    |   movel([0.186644, -1.304676, -2.622886, -0.784827, 1.570796, 1.757440],accel_mss,speed_ms,0,blend_radius_m)
    |   movel([0.187241, -1.304577, -2.622946, -0.784867, 1.570796, 1.758037],accel_mss,speed_ms,0,blend_radius_m)
    |   movel([0.187800, -1.304513, -2.622984, -0.784892, 1.570796, 1.758596],accel_mss,speed_ms,0,blend_radius_m)
    |   movel([0.187953, -1.304694, -2.622875, -0.784820, 1.570796, 1.758749],accel_mss,speed_ms,0,blend_radius_m)
    |   movel([0.187710, -1.304999, -2.622692, -0.784698, 1.570796, 1.758506],accel_mss,speed_ms,0,blend_radius_m)
    |   movel([0.187182, -1.305200, -2.622571, -0.784618, 1.570796, 1.757979],accel_mss,speed_ms,0,blend_radius_m)
    |   movel([0.186600, -1.305390, -2.622457, -0.784543, 1.570796, 1.757397],accel_mss,speed_ms,0,blend_radius_m)
    |   movel([0.185739, -1.305642, -2.622305, -0.784442, 1.570796, 1.756535],accel_mss,speed_ms,0,blend_radius_m)
    |   movel([0.184876, -1.305876, -2.622164, -0.784349, 1.570796, 1.755672],accel_mss,speed_ms,0,blend_radius_m)
    |   movel([0.180549, -1.306967, -2.621506, -0.783916, 1.570796, 1.751345],accel_mss,speed_ms,0,blend_radius_m)
    |   movel([0.180549, -1.272923, -2.604715, -0.834751, 1.570796, 1.751345],accel_mss,speed_ms,0,blend_radius_m)
    |   speed_ms = 1.000
    |   movel([0.180846, -1.271403, -2.605588, -0.835398, 1.570796, 1.751642],accel_mss,speed_ms,0,blend_radius_m)
    |   speed_ms = 0.008
    |   movel([0.180846, -1.299028, -2.619389, -0.793972, 1.570796, 1.751642],accel_mss,speed_ms,0,blend_radius_m)
    |   speed_ms = 0.003
    |   movel([0.180846, -1.302530, -2.621035, -0.788824, 1.570796, 1.751642],accel_mss,speed_ms,0,blend_radius_m)
    |   speed_ms = 0.008
    |   movel([0.176518, -1.303606, -2.620389, -0.788394, 1.570796, 1.747315],accel_mss,speed_ms,0,blend_radius_m)
    |   movel([0.175664, -1.303803, -2.620271, -0.788315, 1.570796, 1.746460],accel_mss,speed_ms,0,blend_radius_m)
    |   movel([0.174818, -1.303978, -2.620165, -0.788245, 1.570796, 1.745615],accel_mss,speed_ms,0,blend_radius_m)
    |   movel([0.174256, -1.304075, -2.620107, -0.788207, 1.570796, 1.745053],accel_mss,speed_ms,0,blend_radius_m)
    |   movel([0.173758, -1.304132, -2.620073, -0.788184, 1.570796, 1.744555],accel_mss,speed_ms,0,blend_radius_m)
    |   movel([0.173618, -1.303922, -2.620199, -0.788268, 1.570796, 1.744415],accel_mss,speed_ms,0,blend_radius_m)
    |   movel([0.173863, -1.303642, -2.620367, -0.788379, 1.570796, 1.744659],accel_mss,speed_ms,0,blend_radius_m)
    |   movel([0.174452, -1.303418, -2.620502, -0.788469, 1.570796, 1.745248],accel_mss,speed_ms,0,blend_radius_m)
    |   movel([0.175069, -1.303213, -2.620625, -0.788551, 1.570796, 1.745865],accel_mss,speed_ms,0,blend_radius_m)
    |   movel([0.175893, -1.302967, -2.620773, -0.788649, 1.570796, 1.746689],accel_mss,speed_ms,0,blend_radius_m)
    |   movel([0.176718, -1.302738, -2.620910, -0.788741, 1.570796, 1.747515],accel_mss,speed_ms,0,blend_radius_m)
    |   movel([0.181025, -1.301632, -2.621573, -0.789184, 1.570796, 1.751821],accel_mss,speed_ms,0,blend_radius_m)
    |   movel([0.185323, -1.300575, -2.622205, -0.789610, 1.570796, 1.756120],accel_mss,speed_ms,0,blend_radius_m)
    |   movel([0.186140, -1.300389, -2.622315, -0.789685, 1.570796, 1.756936],accel_mss,speed_ms,0,blend_radius_m)
    |   movel([0.186952, -1.300226, -2.622412, -0.789750, 1.570796, 1.757748],accel_mss,speed_ms,0,blend_radius_m)
    |   movel([0.187550, -1.300126, -2.622472, -0.789791, 1.570796, 1.758346],accel_mss,speed_ms,0,blend_radius_m)
    |   movel([0.188109, -1.300062, -2.622510, -0.789816, 1.570796, 1.758906],accel_mss,speed_ms,0,blend_radius_m)
    |   movel([0.188263, -1.300243, -2.622402, -0.789743, 1.570796, 1.759059],accel_mss,speed_ms,0,blend_radius_m)
    |   movel([0.188019, -1.300551, -2.622219, -0.789619, 1.570796, 1.758815],accel_mss,speed_ms,0,blend_radius_m)
    |   movel([0.187491, -1.300752, -2.622099, -0.789538, 1.570796, 1.758287],accel_mss,speed_ms,0,blend_radius_m)
    |   movel([0.186908, -1.300943, -2.621985, -0.789461, 1.570796, 1.757704],accel_mss,speed_ms,0,blend_radius_m)
    |   movel([0.186045, -1.301196, -2.621833, -0.789359, 1.570796, 1.756841],accel_mss,speed_ms,0,blend_radius_m)
    |   movel([0.185180, -1.301432, -2.621692, -0.789265, 1.570796, 1.755976],accel_mss,speed_ms,0,blend_radius_m)
    |   movel([0.180846, -1.302530, -2.621035, -0.788824, 1.570796, 1.751642],accel_mss,speed_ms,0,blend_radius_m)
    |   movel([0.180846, -1.305477, -2.622404, -0.784508, 1.570796, 1.751642],accel_mss,speed_ms,0,blend_radius_m)
    |   movel([0.176518, -1.306551, -2.621757, -0.784081, 1.570796, 1.747315],accel_mss,speed_ms,0,blend_radius_m)
    |   movel([0.175664, -1.306747, -2.621638, -0.784003, 1.570796, 1.746460],accel_mss,speed_ms,0,blend_radius_m)
    |   movel([0.174818, -1.306923, -2.621532, -0.783934, 1.570796, 1.745615],accel_mss,speed_ms,0,blend_radius_m)
    |   movel([0.174256, -1.307019, -2.621474, -0.783896, 1.570796, 1.745053],accel_mss,speed_ms,0,blend_radius_m)
    |   movel([0.173758, -1.307076, -2.621440, -0.783873, 1.570796, 1.744555],accel_mss,speed_ms,0,blend_radius_m)
    |   movel([0.173618, -1.306867, -2.621566, -0.783956, 1.570796, 1.744415],accel_mss,speed_ms,0,blend_radius_m)
    |   movel([0.173863, -1.306587, -2.621735, -0.784067, 1.570796, 1.744659],accel_mss,speed_ms,0,blend_radius_m)
    |   movel([0.174452, -1.306364, -2.621870, -0.784155, 1.570796, 1.745248],accel_mss,speed_ms,0,blend_radius_m)
    |   movel([0.175069, -1.306159, -2.621993, -0.784237, 1.570796, 1.745865],accel_mss,speed_ms,0,blend_radius_m)
    |   movel([0.175893, -1.305913, -2.622141, -0.784334, 1.570796, 1.746689],accel_mss,speed_ms,0,blend_radius_m)
    |   movel([0.176718, -1.305685, -2.622279, -0.784425, 1.570796, 1.747515],accel_mss,speed_ms,0,blend_radius_m)
    |   movel([0.181025, -1.304581, -2.622943, -0.784865, 1.570796, 1.751821],accel_mss,speed_ms,0,blend_radius_m)
    |   movel([0.185323, -1.303526, -2.623577, -0.785287, 1.570796, 1.756120],accel_mss,speed_ms,0,blend_radius_m)
    |   movel([0.186140, -1.303340, -2.623688, -0.785361, 1.570796, 1.756936],accel_mss,speed_ms,0,blend_radius_m)
    |   movel([0.186952, -1.303178, -2.623785, -0.785426, 1.570796, 1.757748],accel_mss,speed_ms,0,blend_radius_m)
    |   movel([0.187550, -1.303078, -2.623845, -0.785466, 1.570796, 1.758346],accel_mss,speed_ms,0,blend_radius_m)
    |   movel([0.188109, -1.303014, -2.623883, -0.785492, 1.570796, 1.758906],accel_mss,speed_ms,0,blend_radius_m)
    |   movel([0.188263, -1.303195, -2.623775, -0.785419, 1.570796, 1.759059],accel_mss,speed_ms,0,blend_radius_m)
    |   movel([0.188019, -1.303501, -2.623591, -0.785297, 1.570796, 1.758815],accel_mss,speed_ms,0,blend_radius_m)
    |   movel([0.187491, -1.303702, -2.623471, -0.785216, 1.570796, 1.758287],accel_mss,speed_ms,0,blend_radius_m)
    |   movel([0.186908, -1.303893, -2.623356, -0.785140, 1.570796, 1.757704],accel_mss,speed_ms,0,blend_radius_m)
    |   movel([0.186045, -1.304146, -2.623204, -0.785039, 1.570796, 1.756841],accel_mss,speed_ms,0,blend_radius_m)
    |   movel([0.185180, -1.304381, -2.623063, -0.784945, 1.570796, 1.755976],accel_mss,speed_ms,0,blend_radius_m)
    |   movel([0.180846, -1.305477, -2.622404, -0.784508, 1.570796, 1.751642],accel_mss,speed_ms,0,blend_radius_m)
    |   movel([0.180846, -1.271403, -2.605588, -0.835398, 1.570796, 1.751642],accel_mss,speed_ms,0,blend_radius_m)
    |   speed_ms = 1.000
    |   movel([0.180878, -1.269658, -2.606587, -0.836144, 1.570796, 1.751674],accel_mss,speed_ms,0,blend_radius_m)
    |   speed_ms = 0.008
    |   movel([0.180878, -1.297310, -2.620412, -0.794668, 1.570796, 1.751674],accel_mss,speed_ms,0,blend_radius_m)
    |   speed_ms = 0.003
    |   movel([0.180878, -1.300815, -2.622061, -0.789513, 1.570796, 1.751674],accel_mss,speed_ms,0,blend_radius_m)
    |   speed_ms = 0.008
    |   movel([0.173221, -1.302766, -2.620894, -0.788730, 1.570796, 1.744017],accel_mss,speed_ms,0,blend_radius_m)
    |   movel([0.174123, -1.298088, -2.623685, -0.790616, 1.570796, 1.744920],accel_mss,speed_ms,0,blend_radius_m)
    |   movel([0.174373, -1.296883, -2.624400, -0.791107, 1.570796, 1.745169],accel_mss,speed_ms,0,blend_radius_m)
    |   movel([0.174623, -1.295770, -2.625057, -0.791561, 1.570796, 1.745419],accel_mss,speed_ms,0,blend_radius_m)
    |   movel([0.174967, -1.294373, -2.625881, -0.792134, 1.570796, 1.745763],accel_mss,speed_ms,0,blend_radius_m)
    |   movel([0.175412, -1.293345, -2.626486, -0.792558, 1.570796, 1.746208],accel_mss,speed_ms,0,blend_radius_m)
    |   movel([0.190492, -1.289495, -2.628739, -0.794155, 1.570796, 1.761288],accel_mss,speed_ms,0,blend_radius_m)
    |   movel([0.188541, -1.298906, -2.623199, -0.790284, 1.570796, 1.759338],accel_mss,speed_ms,0,blend_radius_m)
    |   movel([0.180878, -1.300815, -2.622061, -0.789513, 1.570796, 1.751674],accel_mss,speed_ms,0,blend_radius_m)
    |   movel([0.180878, -1.303765, -2.623433, -0.785191, 1.570796, 1.751674],accel_mss,speed_ms,0,blend_radius_m)
    |   movel([0.173221, -1.305712, -2.622262, -0.784414, 1.570796, 1.744017],accel_mss,speed_ms,0,blend_radius_m)
    |   movel([0.174123, -1.301044, -2.625060, -0.786285, 1.570796, 1.744920],accel_mss,speed_ms,0,blend_radius_m)
    |   movel([0.174373, -1.299841, -2.625777, -0.786772, 1.570796, 1.745169],accel_mss,speed_ms,0,blend_radius_m)
    |   movel([0.174623, -1.298730, -2.626436, -0.787222, 1.570796, 1.745419],accel_mss,speed_ms,0,blend_radius_m)
    |   movel([0.174967, -1.297336, -2.627262, -0.787791, 1.570796, 1.745763],accel_mss,speed_ms,0,blend_radius_m)
    |   movel([0.175412, -1.296309, -2.627869, -0.788211, 1.570796, 1.746208],accel_mss,speed_ms,0,blend_radius_m)
    |   movel([0.190492, -1.292466, -2.630127, -0.789796, 1.570796, 1.761288],accel_mss,speed_ms,0,blend_radius_m)
    |   movel([0.188541, -1.301860, -2.624573, -0.785956, 1.570796, 1.759338],accel_mss,speed_ms,0,blend_radius_m)
    |   movel([0.180878, -1.303765, -2.623433, -0.785191, 1.570796, 1.751674],accel_mss,speed_ms,0,blend_radius_m)
    |   movel([0.180878, -1.269658, -2.606587, -0.836144, 1.570796, 1.751674],accel_mss,speed_ms,0,blend_radius_m)
    |   speed_ms = 1.000
    |   movel([0.182720, -1.258496, -2.612890, -0.841002, 1.570796, 1.753516],accel_mss,speed_ms,0,blend_radius_m)
    |   speed_ms = 0.008
    |   movel([0.182720, -1.286315, -2.626867, -0.799207, 1.570796, 1.753516],accel_mss,speed_ms,0,blend_radius_m)
    |   speed_ms = 0.003
    |   movel([0.182720, -1.289844, -2.628536, -0.794009, 1.570796, 1.753516],accel_mss,speed_ms,0,blend_radius_m)
    |   speed_ms = 0.008
    |   movel([0.182439, -1.290140, -2.628363, -0.793886, 1.570796, 1.753235],accel_mss,speed_ms,0,blend_radius_m)
    |   movel([0.182079, -1.290336, -2.628249, -0.793804, 1.570796, 1.752875],accel_mss,speed_ms,0,blend_radius_m)
    |   movel([0.181259, -1.290643, -2.628069, -0.793676, 1.570796, 1.752055],accel_mss,speed_ms,0,blend_radius_m)
    |   movel([0.180843, -1.290767, -2.627997, -0.793625, 1.570796, 1.751639],accel_mss,speed_ms,0,blend_radius_m)
    |   movel([0.179595, -1.291104, -2.627800, -0.793485, 1.570796, 1.750391],accel_mss,speed_ms,0,blend_radius_m)
    |   movel([0.175569, -1.292152, -2.627186, -0.793050, 1.570796, 1.746365],accel_mss,speed_ms,0,blend_radius_m)
    |   movel([0.177282, -1.283292, -2.632329, -0.796768, 1.570796, 1.748078],accel_mss,speed_ms,0,blend_radius_m)
    |   movel([0.181054, -1.282298, -2.632900, -0.797191, 1.570796, 1.751850],accel_mss,speed_ms,0,blend_radius_m)
    |   movel([0.182542, -1.281936, -2.633107, -0.797346, 1.570796, 1.753338],accel_mss,speed_ms,0,blend_radius_m)
    |   movel([0.184186, -1.281601, -2.633299, -0.797489, 1.570796, 1.754982],accel_mss,speed_ms,0,blend_radius_m)
    |   movel([0.184431, -1.281745, -2.633217, -0.797427, 1.570796, 1.755227],accel_mss,speed_ms,0,blend_radius_m)
    |   movel([0.184458, -1.282004, -2.633069, -0.797317, 1.570796, 1.755254],accel_mss,speed_ms,0,blend_radius_m)
    |   movel([0.183920, -1.284771, -2.631478, -0.796141, 1.570796, 1.754716],accel_mss,speed_ms,0,blend_radius_m)
    |   movel([0.183450, -1.287114, -2.630123, -0.795152, 1.570796, 1.754246],accel_mss,speed_ms,0,blend_radius_m)
    |   movel([0.183040, -1.289069, -2.628987, -0.794333, 1.570796, 1.753836],accel_mss,speed_ms,0,blend_radius_m)
    |   movel([0.182907, -1.289456, -2.628762, -0.794171, 1.570796, 1.753704],accel_mss,speed_ms,0,blend_radius_m)
    |   movel([0.182720, -1.289844, -2.628536, -0.794009, 1.570796, 1.753516],accel_mss,speed_ms,0,blend_radius_m)
    |   movel([0.182720, -1.292815, -2.629923, -0.789651, 1.570796, 1.753516],accel_mss,speed_ms,0,blend_radius_m)
    |   movel([0.182439, -1.293111, -2.629750, -0.789529, 1.570796, 1.753235],accel_mss,speed_ms,0,blend_radius_m)
    |   movel([0.182079, -1.293306, -2.629635, -0.789448, 1.570796, 1.752875],accel_mss,speed_ms,0,blend_radius_m)
    |   movel([0.181259, -1.293613, -2.629455, -0.789321, 1.570796, 1.752055],accel_mss,speed_ms,0,blend_radius_m)
    |   movel([0.180843, -1.293736, -2.629383, -0.789270, 1.570796, 1.751639],accel_mss,speed_ms,0,blend_radius_m)
    |   movel([0.179595, -1.294072, -2.629186, -0.789131, 1.570796, 1.750391],accel_mss,speed_ms,0,blend_radius_m)
    |   movel([0.175569, -1.295119, -2.628570, -0.788700, 1.570796, 1.746365],accel_mss,speed_ms,0,blend_radius_m)
    |   movel([0.177282, -1.286275, -2.633726, -0.792388, 1.570796, 1.748078],accel_mss,speed_ms,0,blend_radius_m)
    |   movel([0.181054, -1.285283, -2.634298, -0.792808, 1.570796, 1.751850],accel_mss,speed_ms,0,blend_radius_m)
    |   movel([0.182542, -1.284921, -2.634506, -0.792961, 1.570796, 1.753338],accel_mss,speed_ms,0,blend_radius_m)
    |   movel([0.184186, -1.284587, -2.634699, -0.793104, 1.570796, 1.754982],accel_mss,speed_ms,0,blend_radius_m)
    |   movel([0.184431, -1.284730, -2.634616, -0.793043, 1.570796, 1.755227],accel_mss,speed_ms,0,blend_radius_m)
    |   movel([0.184458, -1.284989, -2.634467, -0.792933, 1.570796, 1.755254],accel_mss,speed_ms,0,blend_radius_m)
    |   movel([0.183920, -1.287751, -2.632873, -0.791766, 1.570796, 1.754716],accel_mss,speed_ms,0,blend_radius_m)
    |   movel([0.183450, -1.290090, -2.631514, -0.790785, 1.570796, 1.754246],accel_mss,speed_ms,0,blend_radius_m)
    |   movel([0.183040, -1.292042, -2.630376, -0.789972, 1.570796, 1.753836],accel_mss,speed_ms,0,blend_radius_m)
    |   movel([0.182907, -1.292427, -2.630150, -0.789812, 1.570796, 1.753704],accel_mss,speed_ms,0,blend_radius_m)
    |   movel([0.182720, -1.292815, -2.629923, -0.789651, 1.570796, 1.753516],accel_mss,speed_ms,0,blend_radius_m)
    |   movel([0.182720, -1.258496, -2.612890, -0.841002, 1.570796, 1.753516],accel_mss,speed_ms,0,blend_radius_m)
    |   speed_ms = 1.000
    |   movel([0.187137, -1.257819, -2.613268, -0.841302, 1.570796, 1.757933],accel_mss,speed_ms,0,blend_radius_m)
    |   speed_ms = 0.008
    |   movel([0.187137, -1.285648, -2.627254, -0.799487, 1.570796, 1.757933],accel_mss,speed_ms,0,blend_radius_m)
    |   speed_ms = 0.003
    |   movel([0.187137, -1.289178, -2.628924, -0.794287, 1.570796, 1.757933],accel_mss,speed_ms,0,blend_radius_m)
    |   speed_ms = 0.008
    |   movel([0.183531, -1.290095, -2.628390, -0.793905, 1.570796, 1.754327],accel_mss,speed_ms,0,blend_radius_m)
    |   movel([0.185413, -1.281310, -2.633466, -0.797613, 1.570796, 1.756210],accel_mss,speed_ms,0,blend_radius_m)
    |   movel([0.189272, -1.280216, -2.634091, -0.798082, 1.570796, 1.760068],accel_mss,speed_ms,0,blend_radius_m)
    |   movel([0.190274, -1.279953, -2.634242, -0.798195, 1.570796, 1.761070],accel_mss,speed_ms,0,blend_radius_m)
    |   movel([0.191233, -1.279720, -2.634374, -0.798294, 1.570796, 1.762029],accel_mss,speed_ms,0,blend_radius_m)
    |   movel([0.191870, -1.279578, -2.634455, -0.798356, 1.570796, 1.762667],accel_mss,speed_ms,0,blend_radius_m)
    |   movel([0.192157, -1.279566, -2.634462, -0.798361, 1.570796, 1.762953],accel_mss,speed_ms,0,blend_radius_m)
    |   movel([0.192312, -1.279706, -2.634382, -0.798301, 1.570796, 1.763109],accel_mss,speed_ms,0,blend_radius_m)
    |   movel([0.192309, -1.280047, -2.634188, -0.798154, 1.570796, 1.763106],accel_mss,speed_ms,0,blend_radius_m)
    |   movel([0.192277, -1.280477, -2.633942, -0.797970, 1.570796, 1.763074],accel_mss,speed_ms,0,blend_radius_m)
    |   movel([0.192200, -1.281060, -2.633609, -0.797720, 1.570796, 1.762997],accel_mss,speed_ms,0,blend_radius_m)
    |   movel([0.192102, -1.281654, -2.633269, -0.797466, 1.570796, 1.762899],accel_mss,speed_ms,0,blend_radius_m)
    |   movel([0.191728, -1.283548, -2.632182, -0.796659, 1.570796, 1.762524],accel_mss,speed_ms,0,blend_radius_m)
    |   movel([0.190747, -1.288270, -2.629452, -0.794667, 1.570796, 1.761543],accel_mss,speed_ms,0,blend_radius_m)
    |   movel([0.187137, -1.289178, -2.628924, -0.794287, 1.570796, 1.757933],accel_mss,speed_ms,0,blend_radius_m)
    |   movel([0.187137, -1.292150, -2.630312, -0.789927, 1.570796, 1.757933],accel_mss,speed_ms,0,blend_radius_m)
    |   movel([0.183531, -1.293065, -2.629777, -0.789547, 1.570796, 1.754327],accel_mss,speed_ms,0,blend_radius_m)
    |   movel([0.185413, -1.284296, -2.634866, -0.793227, 1.570796, 1.756210],accel_mss,speed_ms,0,blend_radius_m)
    |   movel([0.189272, -1.283204, -2.635493, -0.793692, 1.570796, 1.760068],accel_mss,speed_ms,0,blend_radius_m)
    |   movel([0.190274, -1.282941, -2.635643, -0.793804, 1.570796, 1.761070],accel_mss,speed_ms,0,blend_radius_m)
    |   movel([0.191233, -1.282710, -2.635776, -0.793903, 1.570796, 1.762029],accel_mss,speed_ms,0,blend_radius_m)
    |   movel([0.191870, -1.282567, -2.635858, -0.793964, 1.570796, 1.762667],accel_mss,speed_ms,0,blend_radius_m)
    |   movel([0.192157, -1.282556, -2.635864, -0.793969, 1.570796, 1.762953],accel_mss,speed_ms,0,blend_radius_m)
    |   movel([0.192312, -1.282695, -2.635784, -0.793909, 1.570796, 1.763109],accel_mss,speed_ms,0,blend_radius_m)
    |   movel([0.192309, -1.283036, -2.635589, -0.793764, 1.570796, 1.763106],accel_mss,speed_ms,0,blend_radius_m)
    |   movel([0.192277, -1.283465, -2.635343, -0.793581, 1.570796, 1.763074],accel_mss,speed_ms,0,blend_radius_m)
    |   movel([0.192200, -1.284046, -2.635009, -0.793333, 1.570796, 1.762997],accel_mss,speed_ms,0,blend_radius_m)
    |   movel([0.192102, -1.284640, -2.634668, -0.793081, 1.570796, 1.762899],accel_mss,speed_ms,0,blend_radius_m)
    |   movel([0.191728, -1.286531, -2.633578, -0.792280, 1.570796, 1.762524],accel_mss,speed_ms,0,blend_radius_m)
    |   movel([0.190747, -1.291244, -2.630842, -0.790304, 1.570796, 1.761543],accel_mss,speed_ms,0,blend_radius_m)
    |   movel([0.187137, -1.292150, -2.630312, -0.789927, 1.570796, 1.757933],accel_mss,speed_ms,0,blend_radius_m)
    |   movel([0.187137, -1.257819, -2.613268, -0.841302, 1.570796, 1.757933],accel_mss,speed_ms,0,blend_radius_m)
    |   speed_ms = 1.000
    |   movel([0.170291, -1.267997, -2.607535, -0.836857, 1.570796, 1.741087],accel_mss,speed_ms,0,blend_radius_m)
    |   speed_ms = 0.008
    |   movel([0.170291, -1.295674, -2.621382, -0.795333, 1.570796, 1.741087],accel_mss,speed_ms,0,blend_radius_m)
    |   speed_ms = 0.003
    |   movel([0.170291, -1.299183, -2.623034, -0.790172, 1.570796, 1.741087],accel_mss,speed_ms,0,blend_radius_m)
    |   speed_ms = 0.008
    |   movel([0.165114, -1.300395, -2.622312, -0.789682, 1.570796, 1.735911],accel_mss,speed_ms,0,blend_radius_m)
    |   movel([0.162019, -1.301193, -2.621835, -0.789361, 1.570796, 1.732815],accel_mss,speed_ms,0,blend_radius_m)
    |   movel([0.156479, -1.302669, -2.620952, -0.788768, 1.570796, 1.727275],accel_mss,speed_ms,0,blend_radius_m)
    |   movel([0.140820, -1.307018, -2.618332, -0.787039, 1.570796, 1.711616],accel_mss,speed_ms,0,blend_radius_m)
    |   movel([0.140313, -1.310243, -2.616373, -0.785773, 1.570796, 1.711109],accel_mss,speed_ms,0,blend_radius_m)
    |   movel([0.169783, -1.302097, -2.621294, -0.788998, 1.570796, 1.740580],accel_mss,speed_ms,0,blend_radius_m)
    |   movel([0.170156, -1.300617, -2.622179, -0.789593, 1.570796, 1.740953],accel_mss,speed_ms,0,blend_radius_m)
    |   movel([0.170269, -1.300085, -2.622497, -0.789807, 1.570796, 1.741066],accel_mss,speed_ms,0,blend_radius_m)
    |   movel([0.170325, -1.299694, -2.622730, -0.789965, 1.570796, 1.741121],accel_mss,speed_ms,0,blend_radius_m)
    |   movel([0.170347, -1.299327, -2.622948, -0.790114, 1.570796, 1.741143],accel_mss,speed_ms,0,blend_radius_m)
    |   movel([0.170291, -1.302136, -2.624408, -0.785845, 1.570796, 1.741087],accel_mss,speed_ms,0,blend_radius_m)
    |   movel([0.165114, -1.303346, -2.623684, -0.785359, 1.570796, 1.735911],accel_mss,speed_ms,0,blend_radius_m)
    |   movel([0.162019, -1.304143, -2.623206, -0.785040, 1.570796, 1.732815],accel_mss,speed_ms,0,blend_radius_m)
    |   movel([0.156479, -1.305616, -2.622321, -0.784453, 1.570796, 1.727275],accel_mss,speed_ms,0,blend_radius_m)
    |   movel([0.140820, -1.309956, -2.619694, -0.782738, 1.570796, 1.711616],accel_mss,speed_ms,0,blend_radius_m)
    |   movel([0.140313, -1.313175, -2.617731, -0.781483, 1.570796, 1.711109],accel_mss,speed_ms,0,blend_radius_m)
    |   movel([0.169783, -1.305045, -2.622664, -0.784680, 1.570796, 1.740580],accel_mss,speed_ms,0,blend_radius_m)
    |   movel([0.170156, -1.303568, -2.623551, -0.785270, 1.570796, 1.740953],accel_mss,speed_ms,0,blend_radius_m)
    |   movel([0.170269, -1.303037, -2.623869, -0.785483, 1.570796, 1.741066],accel_mss,speed_ms,0,blend_radius_m)
    |   movel([0.170325, -1.302646, -2.624103, -0.785640, 1.570796, 1.741121],accel_mss,speed_ms,0,blend_radius_m)
    |   movel([0.170347, -1.302280, -2.624322, -0.785787, 1.570796, 1.741143],accel_mss,speed_ms,0,blend_radius_m)
    |   movel([0.170291, -1.267997, -2.607535, -0.836857, 1.570796, 1.741087],accel_mss,speed_ms,0,blend_radius_m)
    |   speed_ms = 1.000
    |   movel([0.169563, -1.271947, -2.605276, -0.835166, 1.570796, 1.740360],accel_mss,speed_ms,0,blend_radius_m)
    |   speed_ms = 0.008
    |   movel([0.169563, -1.299564, -2.619069, -0.793756, 1.570796, 1.740360],accel_mss,speed_ms,0,blend_radius_m)
    |   speed_ms = 0.003
    |   movel([0.169563, -1.303064, -2.620715, -0.788610, 1.570796, 1.740360],accel_mss,speed_ms,0,blend_radius_m)
    |   speed_ms = 0.008
    |   movel([0.164403, -1.304267, -2.619992, -0.788130, 1.570796, 1.735200],accel_mss,speed_ms,0,blend_radius_m)
    |   movel([0.161319, -1.305058, -2.619515, -0.787816, 1.570796, 1.732115],accel_mss,speed_ms,0,blend_radius_m)
    |   movel([0.155801, -1.306519, -2.618633, -0.787236, 1.570796, 1.726597],accel_mss,speed_ms,0,blend_radius_m)
    |   movel([0.140190, -1.310831, -2.616014, -0.785544, 1.570796, 1.710986],accel_mss,speed_ms,0,blend_radius_m)
    |   movel([0.139859, -1.314123, -2.613998, -0.784268, 1.570796, 1.710655],accel_mss,speed_ms,0,blend_radius_m)
    |   movel([0.169004, -1.306259, -2.618791, -0.787339, 1.570796, 1.739800],accel_mss,speed_ms,0,blend_radius_m)
    |   movel([0.169404, -1.304628, -2.619774, -0.787986, 1.570796, 1.740201],accel_mss,speed_ms,0,blend_radius_m)
    |   movel([0.169527, -1.304043, -2.620127, -0.788220, 1.570796, 1.740323],accel_mss,speed_ms,0,blend_radius_m)
    |   movel([0.169589, -1.303614, -2.620384, -0.788391, 1.570796, 1.740386],accel_mss,speed_ms,0,blend_radius_m)
    |   movel([0.169620, -1.303200, -2.620633, -0.788556, 1.570796, 1.740417],accel_mss,speed_ms,0,blend_radius_m)
    |   movel([0.169563, -1.306010, -2.622083, -0.784296, 1.570796, 1.740360],accel_mss,speed_ms,0,blend_radius_m)
    |   movel([0.164403, -1.307211, -2.621358, -0.783820, 1.570796, 1.735200],accel_mss,speed_ms,0,blend_radius_m)
    |   movel([0.161319, -1.308000, -2.620881, -0.783508, 1.570796, 1.732115],accel_mss,speed_ms,0,blend_radius_m)
    |   movel([0.155801, -1.309459, -2.619997, -0.782933, 1.570796, 1.726597],accel_mss,speed_ms,0,blend_radius_m)
    |   movel([0.140190, -1.313762, -2.617371, -0.781255, 1.570796, 1.710986],accel_mss,speed_ms,0,blend_radius_m)
    |   movel([0.139859, -1.317048, -2.615350, -0.779991, 1.570796, 1.710655],accel_mss,speed_ms,0,blend_radius_m)
    |   movel([0.169004, -1.309199, -2.620154, -0.783036, 1.570796, 1.739800],accel_mss,speed_ms,0,blend_radius_m)
    |   movel([0.169404, -1.307572, -2.621140, -0.783677, 1.570796, 1.740201],accel_mss,speed_ms,0,blend_radius_m)
    |   movel([0.169527, -1.306987, -2.621494, -0.783908, 1.570796, 1.740323],accel_mss,speed_ms,0,blend_radius_m)
    |   movel([0.169589, -1.306559, -2.621752, -0.784078, 1.570796, 1.740386],accel_mss,speed_ms,0,blend_radius_m)
    |   movel([0.169620, -1.306146, -2.622001, -0.784242, 1.570796, 1.740417],accel_mss,speed_ms,0,blend_radius_m)
    |   movel([0.169563, -1.271947, -2.605276, -0.835166, 1.570796, 1.740360],accel_mss,speed_ms,0,blend_radius_m)
    |   speed_ms = 1.000
    |   movel([0.168841, -1.275879, -2.603009, -0.833501, 1.570796, 1.739637],accel_mss,speed_ms,0,blend_radius_m)
    |   speed_ms = 0.008
    |   movel([0.168841, -1.303435, -2.616748, -0.792206, 1.570796, 1.739637],accel_mss,speed_ms,0,blend_radius_m)
    |   speed_ms = 0.003
    |   movel([0.168841, -1.306926, -2.618387, -0.787076, 1.570796, 1.739637],accel_mss,speed_ms,0,blend_radius_m)
    |   speed_ms = 0.008
    |   movel([0.163710, -1.308113, -2.617668, -0.786608, 1.570796, 1.734506],accel_mss,speed_ms,0,blend_radius_m)
    |   movel([0.160642, -1.308895, -2.617193, -0.786301, 1.570796, 1.731438],accel_mss,speed_ms,0,blend_radius_m)
    |   movel([0.155151, -1.310341, -2.616313, -0.785735, 1.570796, 1.725947],accel_mss,speed_ms,0,blend_radius_m)
    |   movel([0.139630, -1.314604, -2.613702, -0.784083, 1.570796, 1.710426],accel_mss,speed_ms,0,blend_radius_m)
    |   movel([0.139132, -1.317791, -2.611735, -0.782863, 1.570796, 1.709928],accel_mss,speed_ms,0,blend_radius_m)
    |   movel([0.168342, -1.309805, -2.616639, -0.785944, 1.570796, 1.739139],accel_mss,speed_ms,0,blend_radius_m)
    |   movel([0.168710, -1.308344, -2.617528, -0.786517, 1.570796, 1.739506],accel_mss,speed_ms,0,blend_radius_m)
    |   movel([0.168821, -1.307818, -2.617847, -0.786724, 1.570796, 1.739617],accel_mss,speed_ms,0,blend_radius_m)
    |   movel([0.168875, -1.307431, -2.618081, -0.786876, 1.570796, 1.739672],accel_mss,speed_ms,0,blend_radius_m)
    |   movel([0.168897, -1.307069, -2.618301, -0.787019, 1.570796, 1.739693],accel_mss,speed_ms,0,blend_radius_m)
    |   movel([0.168841, -1.309865, -2.619750, -0.782774, 1.570796, 1.739637],accel_mss,speed_ms,0,blend_radius_m)
    |   movel([0.163710, -1.311049, -2.619029, -0.782310, 1.570796, 1.734506],accel_mss,speed_ms,0,blend_radius_m)
    |   movel([0.160642, -1.311830, -2.618553, -0.782006, 1.570796, 1.731438],accel_mss,speed_ms,0,blend_radius_m)
    |   movel([0.155151, -1.313273, -2.617671, -0.781445, 1.570796, 1.725947],accel_mss,speed_ms,0,blend_radius_m)
    |   movel([0.139630, -1.317527, -2.615054, -0.779807, 1.570796, 1.710426],accel_mss,speed_ms,0,blend_radius_m)
    |   movel([0.139132, -1.320708, -2.613082, -0.778599, 1.570796, 1.709928],accel_mss,speed_ms,0,blend_radius_m)
    |   movel([0.168342, -1.312738, -2.617998, -0.781653, 1.570796, 1.739139],accel_mss,speed_ms,0,blend_radius_m)
    |   movel([0.168710, -1.311280, -2.618889, -0.782221, 1.570796, 1.739506],accel_mss,speed_ms,0,blend_radius_m)
    |   movel([0.168821, -1.310755, -2.619208, -0.782426, 1.570796, 1.739617],accel_mss,speed_ms,0,blend_radius_m)
    |   movel([0.168875, -1.310369, -2.619443, -0.782577, 1.570796, 1.739672],accel_mss,speed_ms,0,blend_radius_m)
    |   movel([0.168897, -1.310007, -2.619663, -0.782718, 1.570796, 1.739693],accel_mss,speed_ms,0,blend_radius_m)
    |   movel([0.168841, -1.275879, -2.603009, -0.833501, 1.570796, 1.739637],accel_mss,speed_ms,0,blend_radius_m)
    |   speed_ms = 1.000
    |   movel([0.161956, -1.257077, -2.613681, -0.841631, 1.570796, 1.732752],accel_mss,speed_ms,0,blend_radius_m)
    |   speed_ms = 0.008
    |   movel([0.161956, -1.284916, -2.627678, -0.799795, 1.570796, 1.732752],accel_mss,speed_ms,0,blend_radius_m)
    |   speed_ms = 0.003
    |   movel([0.161956, -1.288448, -2.629349, -0.794593, 1.570796, 1.732752],accel_mss,speed_ms,0,blend_radius_m)
    |   speed_ms = 0.008
    |   movel([0.149359, -1.291972, -2.627292, -0.793125, 1.570796, 1.720155],accel_mss,speed_ms,0,blend_radius_m)
    |   movel([0.154199, -1.263017, -2.643727, -0.805645, 1.570796, 1.724995],accel_mss,speed_ms,0,blend_radius_m)
    |   movel([0.170764, -1.258104, -2.646413, -0.807872, 1.570796, 1.741560],accel_mss,speed_ms,0,blend_radius_m)
    |   movel([0.174686, -1.256990, -2.647018, -0.808381, 1.570796, 1.745482],accel_mss,speed_ms,0,blend_radius_m)
    |   movel([0.179682, -1.255617, -2.647761, -0.809011, 1.570796, 1.750478],accel_mss,speed_ms,0,blend_radius_m)
    |   movel([0.180051, -1.255585, -2.647779, -0.809025, 1.570796, 1.750847],accel_mss,speed_ms,0,blend_radius_m)
    |   movel([0.180204, -1.255831, -2.647645, -0.808912, 1.570796, 1.751000],accel_mss,speed_ms,0,blend_radius_m)
    |   movel([0.179750, -1.258560, -2.646165, -0.807664, 1.570796, 1.750547],accel_mss,speed_ms,0,blend_radius_m)
    |   movel([0.179408, -1.260485, -2.645115, -0.806789, 1.570796, 1.750205],accel_mss,speed_ms,0,blend_radius_m)
    |   movel([0.179047, -1.262413, -2.644059, -0.805917, 1.570796, 1.749843],accel_mss,speed_ms,0,blend_radius_m)
    |   movel([0.177744, -1.269039, -2.640395, -0.802955, 1.570796, 1.748541],accel_mss,speed_ms,0,blend_radius_m)
    |   movel([0.174579, -1.285030, -2.631328, -0.796031, 1.570796, 1.745375],accel_mss,speed_ms,0,blend_radius_m)
    |   movel([0.161956, -1.288448, -2.629349, -0.794593, 1.570796, 1.732752],accel_mss,speed_ms,0,blend_radius_m)
    |   movel([0.161956, -1.291421, -2.630738, -0.790230, 1.570796, 1.732752],accel_mss,speed_ms,0,blend_radius_m)
    |   movel([0.149359, -1.294939, -2.628676, -0.788774, 1.570796, 1.720155],accel_mss,speed_ms,0,blend_radius_m)
    |   movel([0.154199, -1.266035, -2.645153, -0.801201, 1.570796, 1.724995],accel_mss,speed_ms,0,blend_radius_m)
    |   movel([0.170764, -1.261130, -2.647846, -0.803413, 1.570796, 1.741560],accel_mss,speed_ms,0,blend_radius_m)
    |   movel([0.174686, -1.260017, -2.648453, -0.803919, 1.570796, 1.745482],accel_mss,speed_ms,0,blend_radius_m)
    |   movel([0.179682, -1.258647, -2.649198, -0.804544, 1.570796, 1.750478],accel_mss,speed_ms,0,blend_radius_m)
    |   movel([0.180051, -1.258615, -2.649216, -0.804558, 1.570796, 1.750847],accel_mss,speed_ms,0,blend_radius_m)
    |   movel([0.180204, -1.258861, -2.649082, -0.804446, 1.570796, 1.751000],accel_mss,speed_ms,0,blend_radius_m)
    |   movel([0.179750, -1.261585, -2.647598, -0.803206, 1.570796, 1.750547],accel_mss,speed_ms,0,blend_radius_m)
    |   movel([0.179408, -1.263507, -2.646545, -0.802337, 1.570796, 1.750205],accel_mss,speed_ms,0,blend_radius_m)
    |   movel([0.179047, -1.265432, -2.645486, -0.801471, 1.570796, 1.749843],accel_mss,speed_ms,0,blend_radius_m)
    |   movel([0.177744, -1.272046, -2.641813, -0.798530, 1.570796, 1.748541],accel_mss,speed_ms,0,blend_radius_m)
    |   movel([0.174579, -1.288010, -2.632723, -0.791657, 1.570796, 1.745375],accel_mss,speed_ms,0,blend_radius_m)
    |   movel([0.161956, -1.291421, -2.630738, -0.790230, 1.570796, 1.732752],accel_mss,speed_ms,0,blend_radius_m)
    |   movel([0.161956, -1.257077, -2.613681, -0.841631, 1.570796, 1.732752],accel_mss,speed_ms,0,blend_radius_m)
    |   speed_ms = 1.000
    |   movel([0.167427, -1.226250, -2.630272, -0.855867, 1.570796, 1.738223],accel_mss,speed_ms,0,blend_radius_m)
    |   speed_ms = 0.008
    |   movel([0.167427, -1.254505, -2.644693, -0.813190, 1.570796, 1.738223],accel_mss,speed_ms,0,blend_radius_m)
    |   speed_ms = 0.003
    |   movel([0.167427, -1.258098, -2.646416, -0.807875, 1.570796, 1.738223],accel_mss,speed_ms,0,blend_radius_m)
    |   speed_ms = 0.008
    |   movel([0.159713, -1.260325, -2.645202, -0.806861, 1.570796, 1.730509],accel_mss,speed_ms,0,blend_radius_m)
    |   movel([0.158233, -1.260737, -2.644977, -0.806674, 1.570796, 1.729029],accel_mss,speed_ms,0,blend_radius_m)
    |   movel([0.156754, -1.261131, -2.644762, -0.806496, 1.570796, 1.727551],accel_mss,speed_ms,0,blend_radius_m)
    |   movel([0.155748, -1.261384, -2.644623, -0.806382, 1.570796, 1.726544],accel_mss,speed_ms,0,blend_radius_m)
    |   movel([0.154836, -1.261592, -2.644509, -0.806288, 1.570796, 1.725632],accel_mss,speed_ms,0,blend_radius_m)
    |   movel([0.154637, -1.261471, -2.644576, -0.806343, 1.570796, 1.725433],accel_mss,speed_ms,0,blend_radius_m)
    |   movel([0.154743, -1.261182, -2.644734, -0.806473, 1.570796, 1.725539],accel_mss,speed_ms,0,blend_radius_m)
    |   movel([0.155948, -1.260671, -2.645013, -0.806705, 1.570796, 1.726744],accel_mss,speed_ms,0,blend_radius_m)
    |   movel([0.157021, -1.260306, -2.645213, -0.806870, 1.570796, 1.727817],accel_mss,speed_ms,0,blend_radius_m)
    |   movel([0.158464, -1.259840, -2.645468, -0.807082, 1.570796, 1.729261],accel_mss,speed_ms,0,blend_radius_m)
    |   movel([0.159907, -1.259395, -2.645710, -0.807284, 1.570796, 1.730704],accel_mss,speed_ms,0,blend_radius_m)
    |   movel([0.167601, -1.257141, -2.646936, -0.808312, 1.570796, 1.738398],accel_mss,speed_ms,0,blend_radius_m)
    |   movel([0.175296, -1.254958, -2.648117, -0.809313, 1.570796, 1.746093],accel_mss,speed_ms,0,blend_radius_m)
    |   movel([0.176736, -1.254572, -2.648326, -0.809491, 1.570796, 1.747532],accel_mss,speed_ms,0,blend_radius_m)
    |   movel([0.178169, -1.254210, -2.648521, -0.809658, 1.570796, 1.748965],accel_mss,speed_ms,0,blend_radius_m)
    |   movel([0.179227, -1.253961, -2.648655, -0.809773, 1.570796, 1.750023],accel_mss,speed_ms,0,blend_radius_m)
    |   movel([0.180218, -1.253750, -2.648769, -0.809870, 1.570796, 1.751015],accel_mss,speed_ms,0,blend_radius_m)
    |   movel([0.180417, -1.253860, -2.648710, -0.809820, 1.570796, 1.751213],accel_mss,speed_ms,0,blend_radius_m)
    |   movel([0.180318, -1.254157, -2.648550, -0.809683, 1.570796, 1.751115],accel_mss,speed_ms,0,blend_radius_m)
    |   movel([0.179175, -1.254638, -2.648290, -0.809461, 1.570796, 1.749971],accel_mss,speed_ms,0,blend_radius_m)
    |   movel([0.178147, -1.254972, -2.648110, -0.809307, 1.570796, 1.748943],accel_mss,speed_ms,0,blend_radius_m)
    |   movel([0.176647, -1.255436, -2.647859, -0.809094, 1.570796, 1.747443],accel_mss,speed_ms,0,blend_radius_m)
    |   movel([0.175154, -1.255879, -2.647619, -0.808890, 1.570796, 1.745950],accel_mss,speed_ms,0,blend_radius_m)
    |   movel([0.167427, -1.258098, -2.646416, -0.807875, 1.570796, 1.738223],accel_mss,speed_ms,0,blend_radius_m)
    |   movel([0.167427, -1.261124, -2.647850, -0.803416, 1.570796, 1.738223],accel_mss,speed_ms,0,blend_radius_m)
    |   movel([0.159713, -1.263347, -2.646632, -0.802409, 1.570796, 1.730509],accel_mss,speed_ms,0,blend_radius_m)
    |   movel([0.158233, -1.263759, -2.646406, -0.802223, 1.570796, 1.729029],accel_mss,speed_ms,0,blend_radius_m)
    |   movel([0.156754, -1.264152, -2.646191, -0.802046, 1.570796, 1.727551],accel_mss,speed_ms,0,blend_radius_m)
    |   movel([0.155748, -1.264404, -2.646052, -0.801933, 1.570796, 1.726544],accel_mss,speed_ms,0,blend_radius_m)
    |   movel([0.154836, -1.264612, -2.645938, -0.801840, 1.570796, 1.725632],accel_mss,speed_ms,0,blend_radius_m)
    |   movel([0.154637, -1.264491, -2.646004, -0.801894, 1.570796, 1.725433],accel_mss,speed_ms,0,blend_radius_m)
    |   movel([0.154743, -1.264203, -2.646163, -0.802024, 1.570796, 1.725539],accel_mss,speed_ms,0,blend_radius_m)
    |   movel([0.155948, -1.263693, -2.646443, -0.802253, 1.570796, 1.726744],accel_mss,speed_ms,0,blend_radius_m)
    |   movel([0.157021, -1.263328, -2.646643, -0.802418, 1.570796, 1.727817],accel_mss,speed_ms,0,blend_radius_m)
    |   movel([0.158464, -1.262863, -2.646898, -0.802628, 1.570796, 1.729261],accel_mss,speed_ms,0,blend_radius_m)
    |   movel([0.159907, -1.262419, -2.647142, -0.802829, 1.570796, 1.730704],accel_mss,speed_ms,0,blend_radius_m)
    |   movel([0.167601, -1.260168, -2.648371, -0.803850, 1.570796, 1.738398],accel_mss,speed_ms,0,blend_radius_m)
    |   movel([0.175296, -1.257989, -2.649555, -0.804845, 1.570796, 1.746093],accel_mss,speed_ms,0,blend_radius_m)
    |   movel([0.176736, -1.257604, -2.649764, -0.805021, 1.570796, 1.747532],accel_mss,speed_ms,0,blend_radius_m)
    |   movel([0.178169, -1.257242, -2.649960, -0.805187, 1.570796, 1.748965],accel_mss,speed_ms,0,blend_radius_m)
    |   movel([0.179227, -1.256994, -2.650094, -0.805301, 1.570796, 1.750023],accel_mss,speed_ms,0,blend_radius_m)
    |   movel([0.180218, -1.256783, -2.650208, -0.805398, 1.570796, 1.751015],accel_mss,speed_ms,0,blend_radius_m)
    |   movel([0.180417, -1.256893, -2.650149, -0.805347, 1.570796, 1.751213],accel_mss,speed_ms,0,blend_radius_m)
    |   movel([0.180318, -1.257189, -2.649989, -0.805212, 1.570796, 1.751115],accel_mss,speed_ms,0,blend_radius_m)
    |   movel([0.179175, -1.257670, -2.649728, -0.804991, 1.570796, 1.749971],accel_mss,speed_ms,0,blend_radius_m)
    |   movel([0.178147, -1.258002, -2.649548, -0.804839, 1.570796, 1.748943],accel_mss,speed_ms,0,blend_radius_m)
    |   movel([0.176647, -1.258466, -2.649296, -0.804627, 1.570796, 1.747443],accel_mss,speed_ms,0,blend_radius_m)
    |   movel([0.175154, -1.258909, -2.649056, -0.804424, 1.570796, 1.745950],accel_mss,speed_ms,0,blend_radius_m)
    |   movel([0.167427, -1.261124, -2.647850, -0.803416, 1.570796, 1.738223],accel_mss,speed_ms,0,blend_radius_m)
    |   movel([0.167427, -1.226250, -2.630272, -0.855867, 1.570796, 1.738223],accel_mss,speed_ms,0,blend_radius_m)
    |   speed_ms = 1.000
    |   movel([0.167718, -1.224631, -2.631113, -0.856645, 1.570796, 1.738514],accel_mss,speed_ms,0,blend_radius_m)
    |   speed_ms = 0.008
    |   movel([0.167718, -1.252906, -2.645557, -0.813926, 1.570796, 1.738514],accel_mss,speed_ms,0,blend_radius_m)
    |   speed_ms = 0.003
    |   movel([0.167718, -1.256501, -2.647283, -0.808605, 1.570796, 1.738514],accel_mss,speed_ms,0,blend_radius_m)
    |   speed_ms = 0.008
    |   movel([0.159007, -1.259030, -2.645909, -0.807450, 1.570796, 1.729803],accel_mss,speed_ms,0,blend_radius_m)
    |   movel([0.157756, -1.259379, -2.645719, -0.807291, 1.570796, 1.728552],accel_mss,speed_ms,0,blend_radius_m)
    |   movel([0.156516, -1.259698, -2.645545, -0.807146, 1.570796, 1.727312],accel_mss,speed_ms,0,blend_radius_m)
    |   movel([0.155797, -1.259852, -2.645461, -0.807076, 1.570796, 1.726593],accel_mss,speed_ms,0,blend_radius_m)
    |   movel([0.155409, -1.259909, -2.645430, -0.807050, 1.570796, 1.726206],accel_mss,speed_ms,0,blend_radius_m)
    |   movel([0.155039, -1.259911, -2.645428, -0.807049, 1.570796, 1.725836],accel_mss,speed_ms,0,blend_radius_m)
    |   movel([0.154935, -1.259626, -2.645584, -0.807179, 1.570796, 1.725732],accel_mss,speed_ms,0,blend_radius_m)
    |   movel([0.155170, -1.259268, -2.645779, -0.807342, 1.570796, 1.725966],accel_mss,speed_ms,0,blend_radius_m)
    |   movel([0.155640, -1.259018, -2.645916, -0.807456, 1.570796, 1.726436],accel_mss,speed_ms,0,blend_radius_m)
    |   movel([0.156044, -1.258847, -2.646009, -0.807533, 1.570796, 1.726841],accel_mss,speed_ms,0,blend_radius_m)
    |   movel([0.156826, -1.258557, -2.646167, -0.807665, 1.570796, 1.727622],accel_mss,speed_ms,0,blend_radius_m)
    |   movel([0.158038, -1.258155, -2.646385, -0.807849, 1.570796, 1.728834],accel_mss,speed_ms,0,blend_radius_m)
    |   movel([0.159251, -1.257776, -2.646591, -0.808022, 1.570796, 1.730048],accel_mss,speed_ms,0,blend_radius_m)
    |   movel([0.167951, -1.255221, -2.647975, -0.809192, 1.570796, 1.738748],accel_mss,speed_ms,0,blend_radius_m)
    |   movel([0.176656, -1.252744, -2.649310, -0.810335, 1.570796, 1.747452],accel_mss,speed_ms,0,blend_radius_m)
    |   movel([0.177860, -1.252424, -2.649481, -0.810483, 1.570796, 1.748657],accel_mss,speed_ms,0,blend_radius_m)
    |   movel([0.179066, -1.252128, -2.649640, -0.810620, 1.570796, 1.749862],accel_mss,speed_ms,0,blend_radius_m)
    |   movel([0.179828, -1.251973, -2.649724, -0.810693, 1.570796, 1.750624],accel_mss,speed_ms,0,blend_radius_m)
    |   movel([0.180214, -1.251915, -2.649755, -0.810719, 1.570796, 1.751011],accel_mss,speed_ms,0,blend_radius_m)
    |   movel([0.180538, -1.251886, -2.649770, -0.810733, 1.570796, 1.751335],accel_mss,speed_ms,0,blend_radius_m)
    |   movel([0.180764, -1.252051, -2.649681, -0.810656, 1.570796, 1.751561],accel_mss,speed_ms,0,blend_radius_m)
    |   movel([0.180650, -1.252427, -2.649480, -0.810482, 1.570796, 1.751447],accel_mss,speed_ms,0,blend_radius_m)
    |   movel([0.180126, -1.252775, -2.649293, -0.810321, 1.570796, 1.750922],accel_mss,speed_ms,0,blend_radius_m)
    |   movel([0.179717, -1.252948, -2.649200, -0.810241, 1.570796, 1.750513],accel_mss,speed_ms,0,blend_radius_m)
    |   movel([0.178969, -1.253218, -2.649055, -0.810116, 1.570796, 1.749765],accel_mss,speed_ms,0,blend_radius_m)
    |   movel([0.177706, -1.253621, -2.648838, -0.809930, 1.570796, 1.748503],accel_mss,speed_ms,0,blend_radius_m)
    |   movel([0.176447, -1.253997, -2.648636, -0.809756, 1.570796, 1.747243],accel_mss,speed_ms,0,blend_radius_m)
    |   movel([0.167718, -1.256501, -2.647283, -0.808605, 1.570796, 1.738514],accel_mss,speed_ms,0,blend_radius_m)
    |   movel([0.167718, -1.259530, -2.648718, -0.804141, 1.570796, 1.738514],accel_mss,speed_ms,0,blend_radius_m)
    |   movel([0.159007, -1.262054, -2.647341, -0.802994, 1.570796, 1.729803],accel_mss,speed_ms,0,blend_radius_m)
    |   movel([0.157756, -1.262403, -2.647150, -0.802836, 1.570796, 1.728552],accel_mss,speed_ms,0,blend_radius_m)
    |   movel([0.156516, -1.262721, -2.646976, -0.802692, 1.570796, 1.727312],accel_mss,speed_ms,0,blend_radius_m)
    |   movel([0.155797, -1.262875, -2.646892, -0.802623, 1.570796, 1.726593],accel_mss,speed_ms,0,blend_radius_m)
    |   movel([0.155409, -1.262932, -2.646860, -0.802597, 1.570796, 1.726206],accel_mss,speed_ms,0,blend_radius_m)
    |   movel([0.155039, -1.262934, -2.646859, -0.802596, 1.570796, 1.725836],accel_mss,speed_ms,0,blend_radius_m)
    |   movel([0.154935, -1.262650, -2.647015, -0.802724, 1.570796, 1.725732],accel_mss,speed_ms,0,blend_radius_m)
    |   movel([0.155170, -1.262292, -2.647211, -0.802886, 1.570796, 1.725966],accel_mss,speed_ms,0,blend_radius_m)
    |   movel([0.155640, -1.262042, -2.647348, -0.802999, 1.570796, 1.726436],accel_mss,speed_ms,0,blend_radius_m)
    |   movel([0.156044, -1.261872, -2.647441, -0.803076, 1.570796, 1.726841],accel_mss,speed_ms,0,blend_radius_m)
    |   movel([0.156826, -1.261582, -2.647599, -0.803208, 1.570796, 1.727622],accel_mss,speed_ms,0,blend_radius_m)
    |   movel([0.158038, -1.261181, -2.647818, -0.803390, 1.570796, 1.728834],accel_mss,speed_ms,0,blend_radius_m)
    |   movel([0.159251, -1.260802, -2.648025, -0.803562, 1.570796, 1.730048],accel_mss,speed_ms,0,blend_radius_m)
    |   movel([0.167951, -1.258252, -2.649413, -0.804725, 1.570796, 1.738748],accel_mss,speed_ms,0,blend_radius_m)
    |   movel([0.176656, -1.255779, -2.650751, -0.805860, 1.570796, 1.747452],accel_mss,speed_ms,0,blend_radius_m)
    |   movel([0.177860, -1.255459, -2.650923, -0.806007, 1.570796, 1.748657],accel_mss,speed_ms,0,blend_radius_m)
    |   movel([0.179066, -1.255164, -2.651082, -0.806143, 1.570796, 1.749862],accel_mss,speed_ms,0,blend_radius_m)
    |   movel([0.179828, -1.255008, -2.651166, -0.806215, 1.570796, 1.750624],accel_mss,speed_ms,0,blend_radius_m)
    |   movel([0.180214, -1.254951, -2.651197, -0.806241, 1.570796, 1.751011],accel_mss,speed_ms,0,blend_radius_m)
    |   movel([0.180538, -1.254921, -2.651213, -0.806255, 1.570796, 1.751335],accel_mss,speed_ms,0,blend_radius_m)
    |   movel([0.180764, -1.255087, -2.651123, -0.806178, 1.570796, 1.751561],accel_mss,speed_ms,0,blend_radius_m)
    |   movel([0.180650, -1.255462, -2.650921, -0.806006, 1.570796, 1.751447],accel_mss,speed_ms,0,blend_radius_m)
    |   movel([0.180126, -1.255809, -2.650734, -0.805846, 1.570796, 1.750922],accel_mss,speed_ms,0,blend_radius_m)
    |   movel([0.179717, -1.255982, -2.650641, -0.805766, 1.570796, 1.750513],accel_mss,speed_ms,0,blend_radius_m)
    |   movel([0.178969, -1.256252, -2.650495, -0.805642, 1.570796, 1.749765],accel_mss,speed_ms,0,blend_radius_m)
    |   movel([0.177706, -1.256655, -2.650278, -0.805457, 1.570796, 1.748503],accel_mss,speed_ms,0,blend_radius_m)
    |   movel([0.176447, -1.257029, -2.650075, -0.805285, 1.570796, 1.747243],accel_mss,speed_ms,0,blend_radius_m)
    |   movel([0.167718, -1.259530, -2.648718, -0.804141, 1.570796, 1.738514],accel_mss,speed_ms,0,blend_radius_m)
    |   movel([0.167718, -1.224631, -2.631113, -0.856645, 1.570796, 1.738514],accel_mss,speed_ms,0,blend_radius_m)
    |   speed_ms = 1.000
    |   movel([0.168068, -1.222682, -2.632122, -0.857585, 1.570796, 1.738865],accel_mss,speed_ms,0,blend_radius_m)
    |   speed_ms = 0.008
    |   movel([0.168068, -1.250981, -2.646592, -0.814816, 1.570796, 1.738865],accel_mss,speed_ms,0,blend_radius_m)
    |   speed_ms = 0.003
    |   movel([0.168068, -1.254580, -2.648321, -0.809488, 1.570796, 1.738865],accel_mss,speed_ms,0,blend_radius_m)
    |   speed_ms = 0.008
    |   movel([0.159338, -1.257121, -2.646947, -0.808321, 1.570796, 1.730134],accel_mss,speed_ms,0,blend_radius_m)
    |   movel([0.158085, -1.257472, -2.646756, -0.808161, 1.570796, 1.728881],accel_mss,speed_ms,0,blend_radius_m)
    |   movel([0.156842, -1.257793, -2.646582, -0.808014, 1.570796, 1.727638],accel_mss,speed_ms,0,blend_radius_m)
    |   movel([0.156121, -1.257947, -2.646498, -0.807943, 1.570796, 1.726918],accel_mss,speed_ms,0,blend_radius_m)
    |   movel([0.155733, -1.258005, -2.646467, -0.807917, 1.570796, 1.726529],accel_mss,speed_ms,0,blend_radius_m)
    |   movel([0.155362, -1.258008, -2.646465, -0.807916, 1.570796, 1.726158],accel_mss,speed_ms,0,blend_radius_m)
    |   movel([0.155258, -1.257722, -2.646621, -0.808046, 1.570796, 1.726054],accel_mss,speed_ms,0,blend_radius_m)
    |   movel([0.155493, -1.257363, -2.646816, -0.808211, 1.570796, 1.726290],accel_mss,speed_ms,0,blend_radius_m)
    |   movel([0.155964, -1.257111, -2.646952, -0.808326, 1.570796, 1.726760],accel_mss,speed_ms,0,blend_radius_m)
    |   movel([0.156370, -1.256940, -2.647045, -0.808404, 1.570796, 1.727166],accel_mss,speed_ms,0,blend_radius_m)
    |   movel([0.157153, -1.256649, -2.647203, -0.808537, 1.570796, 1.727949],accel_mss,speed_ms,0,blend_radius_m)
    |   movel([0.158367, -1.256245, -2.647422, -0.808723, 1.570796, 1.729164],accel_mss,speed_ms,0,blend_radius_m)
    |   movel([0.159584, -1.255864, -2.647628, -0.808897, 1.570796, 1.730380],accel_mss,speed_ms,0,blend_radius_m)
    |   movel([0.168303, -1.253296, -2.649013, -0.810080, 1.570796, 1.739099],accel_mss,speed_ms,0,blend_radius_m)
    |   movel([0.177027, -1.250806, -2.650348, -0.811234, 1.570796, 1.747823],accel_mss,speed_ms,0,blend_radius_m)
    |   movel([0.178233, -1.250485, -2.650520, -0.811384, 1.570796, 1.749030],accel_mss,speed_ms,0,blend_radius_m)
    |   movel([0.179441, -1.250187, -2.650679, -0.811522, 1.570796, 1.750238],accel_mss,speed_ms,0,blend_radius_m)
    |   movel([0.180205, -1.250031, -2.650763, -0.811595, 1.570796, 1.751001],accel_mss,speed_ms,0,blend_radius_m)
    |   movel([0.180593, -1.249973, -2.650794, -0.811622, 1.570796, 1.751389],accel_mss,speed_ms,0,blend_radius_m)
    |   movel([0.180917, -1.249943, -2.650810, -0.811636, 1.570796, 1.751714],accel_mss,speed_ms,0,blend_radius_m)
    |   movel([0.181144, -1.250109, -2.650721, -0.811559, 1.570796, 1.751940],accel_mss,speed_ms,0,blend_radius_m)
    |   movel([0.181029, -1.250486, -2.650520, -0.811383, 1.570796, 1.751826],accel_mss,speed_ms,0,blend_radius_m)
    |   movel([0.180504, -1.250835, -2.650333, -0.811221, 1.570796, 1.751300],accel_mss,speed_ms,0,blend_radius_m)
    |   movel([0.180094, -1.251009, -2.650240, -0.811140, 1.570796, 1.750890],accel_mss,speed_ms,0,blend_radius_m)
    |   movel([0.179344, -1.251281, -2.650095, -0.811014, 1.570796, 1.750140],accel_mss,speed_ms,0,blend_radius_m)
    |   movel([0.178079, -1.251686, -2.649878, -0.810826, 1.570796, 1.748875],accel_mss,speed_ms,0,blend_radius_m)
    |   movel([0.176816, -1.252063, -2.649675, -0.810651, 1.570796, 1.747613],accel_mss,speed_ms,0,blend_radius_m)
    |   movel([0.168068, -1.254580, -2.648321, -0.809488, 1.570796, 1.738865],accel_mss,speed_ms,0,blend_radius_m)
    |   movel([0.168068, -1.257612, -2.649760, -0.805018, 1.570796, 1.738865],accel_mss,speed_ms,0,blend_radius_m)
    |   movel([0.159338, -1.260149, -2.648381, -0.803859, 1.570796, 1.730134],accel_mss,speed_ms,0,blend_radius_m)
    |   movel([0.158085, -1.260499, -2.648191, -0.803700, 1.570796, 1.728881],accel_mss,speed_ms,0,blend_radius_m)
    |   movel([0.156842, -1.260819, -2.648016, -0.803554, 1.570796, 1.727638],accel_mss,speed_ms,0,blend_radius_m)
    |   movel([0.156121, -1.260973, -2.647932, -0.803484, 1.570796, 1.726918],accel_mss,speed_ms,0,blend_radius_m)
    |   movel([0.155733, -1.261031, -2.647900, -0.803458, 1.570796, 1.726529],accel_mss,speed_ms,0,blend_radius_m)
    |   movel([0.155362, -1.261034, -2.647899, -0.803456, 1.570796, 1.726158],accel_mss,speed_ms,0,blend_radius_m)
    |   movel([0.155258, -1.260749, -2.648054, -0.803586, 1.570796, 1.726054],accel_mss,speed_ms,0,blend_radius_m)
    |   movel([0.155493, -1.260390, -2.648250, -0.803749, 1.570796, 1.726290],accel_mss,speed_ms,0,blend_radius_m)
    |   movel([0.155964, -1.260139, -2.648387, -0.803863, 1.570796, 1.726760],accel_mss,speed_ms,0,blend_radius_m)
    |   movel([0.156370, -1.259968, -2.648480, -0.803941, 1.570796, 1.727166],accel_mss,speed_ms,0,blend_radius_m)
    |   movel([0.157153, -1.259677, -2.648638, -0.804074, 1.570796, 1.727949],accel_mss,speed_ms,0,blend_radius_m)
    |   movel([0.158367, -1.259273, -2.648858, -0.804258, 1.570796, 1.729164],accel_mss,speed_ms,0,blend_radius_m)
    |   movel([0.159584, -1.258893, -2.649065, -0.804431, 1.570796, 1.730380],accel_mss,speed_ms,0,blend_radius_m)
    |   movel([0.168303, -1.256330, -2.650453, -0.805606, 1.570796, 1.739099],accel_mss,speed_ms,0,blend_radius_m)
    |   movel([0.177027, -1.253844, -2.651792, -0.806753, 1.570796, 1.747823],accel_mss,speed_ms,0,blend_radius_m)
    |   movel([0.178233, -1.253523, -2.651965, -0.806902, 1.570796, 1.749030],accel_mss,speed_ms,0,blend_radius_m)
    |   movel([0.179441, -1.253226, -2.652124, -0.807039, 1.570796, 1.750238],accel_mss,speed_ms,0,blend_radius_m)
    |   movel([0.180205, -1.253070, -2.652208, -0.807112, 1.570796, 1.751001],accel_mss,speed_ms,0,blend_radius_m)
    |   movel([0.180593, -1.253012, -2.652239, -0.807138, 1.570796, 1.751389],accel_mss,speed_ms,0,blend_radius_m)
    |   movel([0.180917, -1.252982, -2.652255, -0.807152, 1.570796, 1.751714],accel_mss,speed_ms,0,blend_radius_m)
    |   movel([0.181144, -1.253148, -2.652166, -0.807075, 1.570796, 1.751940],accel_mss,speed_ms,0,blend_radius_m)
    |   movel([0.181029, -1.253524, -2.651964, -0.806901, 1.570796, 1.751826],accel_mss,speed_ms,0,blend_radius_m)
    |   movel([0.180504, -1.253872, -2.651777, -0.806740, 1.570796, 1.751300],accel_mss,speed_ms,0,blend_radius_m)
    |   movel([0.180094, -1.254046, -2.651684, -0.806659, 1.570796, 1.750890],accel_mss,speed_ms,0,blend_radius_m)
    |   movel([0.179344, -1.254317, -2.651538, -0.806534, 1.570796, 1.750140],accel_mss,speed_ms,0,blend_radius_m)
    |   movel([0.178079, -1.254722, -2.651320, -0.806347, 1.570796, 1.748875],accel_mss,speed_ms,0,blend_radius_m)
    |   movel([0.176816, -1.255099, -2.651117, -0.806173, 1.570796, 1.747613],accel_mss,speed_ms,0,blend_radius_m)
    |   movel([0.168068, -1.257612, -2.649760, -0.805018, 1.570796, 1.738865],accel_mss,speed_ms,0,blend_radius_m)
    |   movel([0.168068, -1.222682, -2.632122, -0.857585, 1.570796, 1.738865],accel_mss,speed_ms,0,blend_radius_m)
    |   speed_ms = 1.000
    |   movel([0.168420, -1.220727, -2.633129, -0.858533, 1.570796, 1.739217],accel_mss,speed_ms,0,blend_radius_m)
    |   speed_ms = 0.008
    |   movel([0.168420, -1.249050, -2.647626, -0.815713, 1.570796, 1.739217],accel_mss,speed_ms,0,blend_radius_m)
    |   speed_ms = 0.003
    |   movel([0.168420, -1.252653, -2.649359, -0.810377, 1.570796, 1.739217],accel_mss,speed_ms,0,blend_radius_m)
    |   speed_ms = 0.008
    |   movel([0.160658, -1.254912, -2.648142, -0.809335, 1.570796, 1.731454],accel_mss,speed_ms,0,blend_radius_m)
    |   movel([0.159169, -1.255330, -2.647916, -0.809142, 1.570796, 1.729966],accel_mss,speed_ms,0,blend_radius_m)
    |   movel([0.157681, -1.255730, -2.647700, -0.808959, 1.570796, 1.728478],accel_mss,speed_ms,0,blend_radius_m)
    |   movel([0.156669, -1.255986, -2.647562, -0.808841, 1.570796, 1.727465],accel_mss,speed_ms,0,blend_radius_m)
    |   movel([0.155751, -1.256198, -2.647447, -0.808744, 1.570796, 1.726548],accel_mss,speed_ms,0,blend_radius_m)
    |   movel([0.155551, -1.256076, -2.647513, -0.808800, 1.570796, 1.726347],accel_mss,speed_ms,0,blend_radius_m)
    |   movel([0.155658, -1.255784, -2.647671, -0.808934, 1.570796, 1.726454],accel_mss,speed_ms,0,blend_radius_m)
    |   movel([0.156871, -1.255267, -2.647950, -0.809171, 1.570796, 1.727667],accel_mss,speed_ms,0,blend_radius_m)
    |   movel([0.157950, -1.254897, -2.648150, -0.809341, 1.570796, 1.728747],accel_mss,speed_ms,0,blend_radius_m)
    |   movel([0.159403, -1.254425, -2.648405, -0.809559, 1.570796, 1.730199],accel_mss,speed_ms,0,blend_radius_m)
    |   movel([0.160855, -1.253974, -2.648648, -0.809767, 1.570796, 1.731651],accel_mss,speed_ms,0,blend_radius_m)
    |   movel([0.168597, -1.251687, -2.649877, -0.810825, 1.570796, 1.739393],accel_mss,speed_ms,0,blend_radius_m)
    |   movel([0.176340, -1.249473, -2.651060, -0.811855, 1.570796, 1.747136],accel_mss,speed_ms,0,blend_radius_m)
    |   movel([0.177788, -1.249082, -2.651269, -0.812038, 1.570796, 1.748585],accel_mss,speed_ms,0,blend_radius_m)
    |   movel([0.179230, -1.248714, -2.651465, -0.812210, 1.570796, 1.750026],accel_mss,speed_ms,0,blend_radius_m)
    |   movel([0.180295, -1.248461, -2.651599, -0.812328, 1.570796, 1.751091],accel_mss,speed_ms,0,blend_radius_m)
    |   movel([0.181292, -1.248247, -2.651713, -0.812429, 1.570796, 1.752089],accel_mss,speed_ms,0,blend_radius_m)
    |   movel([0.181492, -1.248357, -2.651655, -0.812377, 1.570796, 1.752288],accel_mss,speed_ms,0,blend_radius_m)
    |   movel([0.181392, -1.248656, -2.651496, -0.812237, 1.570796, 1.752189],accel_mss,speed_ms,0,blend_radius_m)
    |   movel([0.180241, -1.249144, -2.651236, -0.812009, 1.570796, 1.751037],accel_mss,speed_ms,0,blend_radius_m)
    |   movel([0.179207, -1.249482, -2.651056, -0.811851, 1.570796, 1.750003],accel_mss,speed_ms,0,blend_radius_m)
    |   movel([0.177698, -1.249953, -2.650804, -0.811632, 1.570796, 1.748494],accel_mss,speed_ms,0,blend_radius_m)
    |   movel([0.176196, -1.250403, -2.650564, -0.811422, 1.570796, 1.746992],accel_mss,speed_ms,0,blend_radius_m)
    |   movel([0.168420, -1.252653, -2.649359, -0.810377, 1.570796, 1.739217],accel_mss,speed_ms,0,blend_radius_m)
    |   movel([0.168420, -1.255688, -2.650800, -0.805902, 1.570796, 1.739217],accel_mss,speed_ms,0,blend_radius_m)
    |   movel([0.160658, -1.257943, -2.649580, -0.804866, 1.570796, 1.731454],accel_mss,speed_ms,0,blend_radius_m)
    |   movel([0.159169, -1.258361, -2.649354, -0.804675, 1.570796, 1.729966],accel_mss,speed_ms,0,blend_radius_m)
    |   movel([0.157681, -1.258759, -2.649137, -0.804492, 1.570796, 1.728478],accel_mss,speed_ms,0,blend_radius_m)
    |   movel([0.156669, -1.259016, -2.648998, -0.804375, 1.570796, 1.727465],accel_mss,speed_ms,0,blend_radius_m)
    |   movel([0.155751, -1.259226, -2.648883, -0.804279, 1.570796, 1.726548],accel_mss,speed_ms,0,blend_radius_m)
    |   movel([0.155551, -1.259105, -2.648949, -0.804335, 1.570796, 1.726347],accel_mss,speed_ms,0,blend_radius_m)
    |   movel([0.155658, -1.258814, -2.649107, -0.804468, 1.570796, 1.726454],accel_mss,speed_ms,0,blend_radius_m)
    |   movel([0.156871, -1.258298, -2.649388, -0.804703, 1.570796, 1.727667],accel_mss,speed_ms,0,blend_radius_m)
    |   movel([0.157950, -1.257928, -2.649588, -0.804873, 1.570796, 1.728747],accel_mss,speed_ms,0,blend_radius_m)
    |   movel([0.159403, -1.257456, -2.649844, -0.805089, 1.570796, 1.730199],accel_mss,speed_ms,0,blend_radius_m)
    |   movel([0.160855, -1.257006, -2.650088, -0.805295, 1.570796, 1.731651],accel_mss,speed_ms,0,blend_radius_m)
    |   movel([0.168597, -1.254723, -2.651319, -0.806346, 1.570796, 1.739393],accel_mss,speed_ms,0,blend_radius_m)
    |   movel([0.176340, -1.252513, -2.652506, -0.807370, 1.570796, 1.747136],accel_mss,speed_ms,0,blend_radius_m)
    |   movel([0.177788, -1.252122, -2.652715, -0.807552, 1.570796, 1.748585],accel_mss,speed_ms,0,blend_radius_m)
    |   movel([0.179230, -1.251755, -2.652912, -0.807723, 1.570796, 1.750026],accel_mss,speed_ms,0,blend_radius_m)
    |   movel([0.180295, -1.251503, -2.653047, -0.807840, 1.570796, 1.751091],accel_mss,speed_ms,0,blend_radius_m)
    |   movel([0.181292, -1.251288, -2.653161, -0.807940, 1.570796, 1.752089],accel_mss,speed_ms,0,blend_radius_m)
    |   movel([0.181492, -1.251399, -2.653102, -0.807888, 1.570796, 1.752288],accel_mss,speed_ms,0,blend_radius_m)
    |   movel([0.181392, -1.251697, -2.652942, -0.807749, 1.570796, 1.752189],accel_mss,speed_ms,0,blend_radius_m)
    |   movel([0.180241, -1.252184, -2.652682, -0.807523, 1.570796, 1.751037],accel_mss,speed_ms,0,blend_radius_m)
    |   movel([0.179207, -1.252522, -2.652501, -0.807366, 1.570796, 1.750003],accel_mss,speed_ms,0,blend_radius_m)
    |   movel([0.177698, -1.252992, -2.652250, -0.807148, 1.570796, 1.748494],accel_mss,speed_ms,0,blend_radius_m)
    |   movel([0.176196, -1.253441, -2.652009, -0.806940, 1.570796, 1.746992],accel_mss,speed_ms,0,blend_radius_m)
    |   movel([0.168420, -1.255688, -2.650800, -0.805902, 1.570796, 1.739217],accel_mss,speed_ms,0,blend_radius_m)
    |   movel([0.168420, -1.220727, -2.633129, -0.858533, 1.570796, 1.739217],accel_mss,speed_ms,0,blend_radius_m)
    |   speed_ms = 1.000
    |   movel([0.168875, -1.218663, -2.634188, -0.859538, 1.570796, 1.739671],accel_mss,speed_ms,0,blend_radius_m)
    |   speed_ms = 0.008
    |   movel([0.168875, -1.247010, -2.648714, -0.816665, 1.570796, 1.739671],accel_mss,speed_ms,0,blend_radius_m)
    |   speed_ms = 0.003
    |   movel([0.168875, -1.250617, -2.650450, -0.811322, 1.570796, 1.739671],accel_mss,speed_ms,0,blend_radius_m)
    |   speed_ms = 0.008
    |   movel([0.155650, -1.254449, -2.648392, -0.809548, 1.570796, 1.726446],accel_mss,speed_ms,0,blend_radius_m)
    |   movel([0.159260, -1.233332, -2.659514, -0.819543, 1.570796, 1.730057],accel_mss,speed_ms,0,blend_radius_m)
    |   movel([0.174647, -1.228553, -2.661958, -0.821878, 1.570796, 1.745443],accel_mss,speed_ms,0,blend_radius_m)
    |   movel([0.178415, -1.227420, -2.662534, -0.822435, 1.570796, 1.749212],accel_mss,speed_ms,0,blend_radius_m)
    |   movel([0.181652, -1.226472, -2.663014, -0.822903, 1.570796, 1.752448],accel_mss,speed_ms,0,blend_radius_m)
    |   movel([0.185675, -1.225319, -2.663598, -0.823473, 1.570796, 1.756471],accel_mss,speed_ms,0,blend_radius_m)
    |   movel([0.185993, -1.225295, -2.663609, -0.823485, 1.570796, 1.756789],accel_mss,speed_ms,0,blend_radius_m)
    |   movel([0.186154, -1.225455, -2.663529, -0.823406, 1.570796, 1.756950],accel_mss,speed_ms,0,blend_radius_m)
    |   movel([0.185931, -1.227069, -2.662712, -0.822608, 1.570796, 1.756727],accel_mss,speed_ms,0,blend_radius_m)
    |   movel([0.185666, -1.228682, -2.661893, -0.821815, 1.570796, 1.756463],accel_mss,speed_ms,0,blend_radius_m)
    |   movel([0.185378, -1.230305, -2.661065, -0.821019, 1.570796, 1.756174],accel_mss,speed_ms,0,blend_radius_m)
    |   movel([0.184441, -1.235136, -2.658584, -0.818669, 1.570796, 1.755237],accel_mss,speed_ms,0,blend_radius_m)
    |   movel([0.182126, -1.246905, -2.652426, -0.813058, 1.570796, 1.752922],accel_mss,speed_ms,0,blend_radius_m)
    |   movel([0.168875, -1.250617, -2.650450, -0.811322, 1.570796, 1.739671],accel_mss,speed_ms,0,blend_radius_m)
    |   movel([0.168875, -1.253654, -2.651894, -0.806841, 1.570796, 1.739671],accel_mss,speed_ms,0,blend_radius_m)
    |   movel([0.155650, -1.257481, -2.649831, -0.805078, 1.570796, 1.726446],accel_mss,speed_ms,0,blend_radius_m)
    |   movel([0.159260, -1.236396, -2.660983, -0.815010, 1.570796, 1.730057],accel_mss,speed_ms,0,blend_radius_m)
    |   movel([0.174647, -1.231623, -2.663434, -0.817331, 1.570796, 1.745443],accel_mss,speed_ms,0,blend_radius_m)
    |   movel([0.178415, -1.230492, -2.664011, -0.817885, 1.570796, 1.749212],accel_mss,speed_ms,0,blend_radius_m)
    |   movel([0.181652, -1.229546, -2.664493, -0.818350, 1.570796, 1.752448],accel_mss,speed_ms,0,blend_radius_m)
    |   movel([0.185675, -1.228394, -2.665078, -0.818917, 1.570796, 1.756471],accel_mss,speed_ms,0,blend_radius_m)
    |   movel([0.185993, -1.228370, -2.665090, -0.818929, 1.570796, 1.756789],accel_mss,speed_ms,0,blend_radius_m)
    |   movel([0.186154, -1.228530, -2.665009, -0.818850, 1.570796, 1.756950],accel_mss,speed_ms,0,blend_radius_m)
    |   movel([0.185931, -1.230142, -2.664190, -0.818057, 1.570796, 1.756727],accel_mss,speed_ms,0,blend_radius_m)
    |   movel([0.185666, -1.231752, -2.663368, -0.817268, 1.570796, 1.756463],accel_mss,speed_ms,0,blend_radius_m)
    |   movel([0.185378, -1.233373, -2.662539, -0.816477, 1.570796, 1.756174],accel_mss,speed_ms,0,blend_radius_m)
    |   movel([0.184441, -1.238197, -2.660051, -0.814141, 1.570796, 1.755237],accel_mss,speed_ms,0,blend_radius_m)
    |   movel([0.182126, -1.249948, -2.653876, -0.808565, 1.570796, 1.752922],accel_mss,speed_ms,0,blend_radius_m)
    |   movel([0.168875, -1.253654, -2.651894, -0.806841, 1.570796, 1.739671],accel_mss,speed_ms,0,blend_radius_m)
    |   movel([0.168875, -1.218663, -2.634188, -0.859538, 1.570796, 1.739671],accel_mss,speed_ms,0,blend_radius_m)
    |   speed_ms = 1.000
    |   movel([0.173307, -1.195696, -2.645650, -0.871043, 1.570796, 1.744104],accel_mss,speed_ms,0,blend_radius_m)
    |   speed_ms = 0.008
    |   movel([0.173307, -1.224299, -2.660493, -0.827598, 1.570796, 1.744104],accel_mss,speed_ms,0,blend_radius_m)
    |   speed_ms = 0.003
    |   movel([0.173307, -1.227944, -2.662268, -0.822177, 1.570796, 1.744104],accel_mss,speed_ms,0,blend_radius_m)
    |   speed_ms = 0.008
    |   movel([0.159992, -1.232010, -2.660193, -0.820186, 1.570796, 1.730788],accel_mss,speed_ms,0,blend_radius_m)
    |   movel([0.162021, -1.220313, -2.666111, -0.825965, 1.570796, 1.732817],accel_mss,speed_ms,0,blend_radius_m)
    |   movel([0.189040, -1.212048, -2.670198, -0.830142, 1.570796, 1.759836],accel_mss,speed_ms,0,blend_radius_m)
    |   movel([0.186654, -1.223994, -2.664265, -0.824129, 1.570796, 1.757450],accel_mss,speed_ms,0,blend_radius_m)
    |   movel([0.173307, -1.227944, -2.662268, -0.822177, 1.570796, 1.744104],accel_mss,speed_ms,0,blend_radius_m)
    |   movel([0.173307, -1.231015, -2.663745, -0.817629, 1.570796, 1.744104],accel_mss,speed_ms,0,blend_radius_m)
    |   movel([0.159992, -1.235075, -2.661664, -0.815650, 1.570796, 1.730788],accel_mss,speed_ms,0,blend_radius_m)
    |   movel([0.162021, -1.223395, -2.667599, -0.821395, 1.570796, 1.732817],accel_mss,speed_ms,0,blend_radius_m)
    |   movel([0.189040, -1.215141, -2.671698, -0.825550, 1.570796, 1.759836],accel_mss,speed_ms,0,blend_radius_m)
    |   movel([0.186654, -1.227071, -2.665748, -0.819570, 1.570796, 1.757450],accel_mss,speed_ms,0,blend_radius_m)
    |   movel([0.173307, -1.231015, -2.663745, -0.817629, 1.570796, 1.744104],accel_mss,speed_ms,0,blend_radius_m)
    |   movel([0.173307, -1.195696, -2.645650, -0.871043, 1.570796, 1.744104],accel_mss,speed_ms,0,blend_radius_m)
    |   speed_ms = 1.000
    |   movel([0.143176, -1.205189, -2.640983, -0.866217, 1.570796, 1.713973],accel_mss,speed_ms,0,blend_radius_m)
    |   speed_ms = 0.008
    |   movel([0.143176, -1.233691, -2.655695, -0.823004, 1.570796, 1.713973],accel_mss,speed_ms,0,blend_radius_m)
    |   speed_ms = 0.003
    |   movel([0.143176, -1.237320, -2.657454, -0.817615, 1.570796, 1.713973],accel_mss,speed_ms,0,blend_radius_m)
    |   speed_ms = 0.008
    |   movel([0.129946, -1.241634, -2.655204, -0.815551, 1.570796, 1.700743],accel_mss,speed_ms,0,blend_radius_m)
    |   movel([0.131578, -1.230231, -2.661103, -0.821055, 1.570796, 1.702374],accel_mss,speed_ms,0,blend_radius_m)
    |   movel([0.158429, -1.221450, -2.665542, -0.825396, 1.570796, 1.729225],accel_mss,speed_ms,0,blend_radius_m)
    |   movel([0.156447, -1.233113, -2.659626, -0.819650, 1.570796, 1.727243],accel_mss,speed_ms,0,blend_radius_m)
    |   movel([0.143176, -1.237320, -2.657454, -0.817615, 1.570796, 1.713973],accel_mss,speed_ms,0,blend_radius_m)
    |   movel([0.143176, -1.240378, -2.658917, -0.813094, 1.570796, 1.713973],accel_mss,speed_ms,0,blend_radius_m)
    |   movel([0.129946, -1.244686, -2.656661, -0.811042, 1.570796, 1.700743],accel_mss,speed_ms,0,blend_radius_m)
    |   movel([0.131578, -1.233299, -2.662577, -0.816513, 1.570796, 1.702374],accel_mss,speed_ms,0,blend_radius_m)
    |   movel([0.158429, -1.224531, -2.667029, -0.820830, 1.570796, 1.729225],accel_mss,speed_ms,0,blend_radius_m)
    |   movel([0.156447, -1.236177, -2.661096, -0.815116, 1.570796, 1.727243],accel_mss,speed_ms,0,blend_radius_m)
    |   movel([0.143176, -1.240378, -2.658917, -0.813094, 1.570796, 1.713973],accel_mss,speed_ms,0,blend_radius_m)
    |   movel([0.143176, -1.205189, -2.640983, -0.866217, 1.570796, 1.713973],accel_mss,speed_ms,0,blend_radius_m)
    |   speed_ms = 1.000
    |   movel([0.139920, -1.227582, -2.629578, -0.855229, 1.570796, 1.710717],accel_mss,speed_ms,0,blend_radius_m)
    |   speed_ms = 0.008
    |   movel([0.139920, -1.255820, -2.643981, -0.812588, 1.570796, 1.710717],accel_mss,speed_ms,0,blend_radius_m)
    |   speed_ms = 0.003
    |   movel([0.139920, -1.259410, -2.645702, -0.807277, 1.570796, 1.710717],accel_mss,speed_ms,0,blend_radius_m)
    |   speed_ms = 0.008
    |   movel([0.126505, -1.263647, -2.643381, -0.805361, 1.570796, 1.697301],accel_mss,speed_ms,0,blend_radius_m)
    |   movel([0.129457, -1.242718, -2.654635, -0.815035, 1.570796, 1.700253],accel_mss,speed_ms,0,blend_radius_m)
    |   movel([0.156987, -1.233882, -2.659231, -0.819276, 1.570796, 1.727783],accel_mss,speed_ms,0,blend_radius_m)
    |   movel([0.153376, -1.255285, -2.647941, -0.809163, 1.570796, 1.724173],accel_mss,speed_ms,0,blend_radius_m)
    |   movel([0.139920, -1.259410, -2.645702, -0.807277, 1.570796, 1.710717],accel_mss,speed_ms,0,blend_radius_m)
    |   movel([0.139920, -1.262434, -2.647133, -0.802822, 1.570796, 1.710717],accel_mss,speed_ms,0,blend_radius_m)
    |   movel([0.126505, -1.266664, -2.644806, -0.800919, 1.570796, 1.697301],accel_mss,speed_ms,0,blend_radius_m)
    |   movel([0.129457, -1.245768, -2.656091, -0.810530, 1.570796, 1.700253],accel_mss,speed_ms,0,blend_radius_m)
    |   movel([0.156987, -1.236945, -2.660699, -0.814745, 1.570796, 1.727783],accel_mss,speed_ms,0,blend_radius_m)
    |   movel([0.153376, -1.258315, -2.649378, -0.804695, 1.570796, 1.724173],accel_mss,speed_ms,0,blend_radius_m)
    |   movel([0.139920, -1.262434, -2.647133, -0.802822, 1.570796, 1.710717],accel_mss,speed_ms,0,blend_radius_m)
    |   movel([0.139920, -1.227582, -2.629578, -0.855229, 1.570796, 1.710717],accel_mss,speed_ms,0,blend_radius_m)
    |   speed_ms = 1.000
    |   movel([0.139630, -1.229499, -2.628575, -0.854315, 1.570796, 1.710426],accel_mss,speed_ms,0,blend_radius_m)
    |   speed_ms = 0.008
    |   movel([0.139630, -1.257714, -2.642952, -0.811724, 1.570796, 1.710426],accel_mss,speed_ms,0,blend_radius_m)
    |   speed_ms = 0.003
    |   movel([0.139630, -1.261300, -2.644669, -0.806420, 1.570796, 1.710426],accel_mss,speed_ms,0,blend_radius_m)
    |   speed_ms = 0.008
    |   movel([0.133490, -1.263196, -2.643629, -0.805564, 1.570796, 1.704286],accel_mss,speed_ms,0,blend_radius_m)
    |   movel([0.129732, -1.264323, -2.643008, -0.805057, 1.570796, 1.700529],accel_mss,speed_ms,0,blend_radius_m)
    |   movel([0.126757, -1.265196, -2.642527, -0.804666, 1.570796, 1.697554],accel_mss,speed_ms,0,blend_radius_m)
    |   movel([0.126686, -1.264981, -2.642646, -0.804763, 1.570796, 1.697483],accel_mss,speed_ms,0,blend_radius_m)
    |   movel([0.130079, -1.263774, -2.643311, -0.805304, 1.570796, 1.700875],accel_mss,speed_ms,0,blend_radius_m)
    |   movel([0.133684, -1.262580, -2.643967, -0.805842, 1.570796, 1.704480],accel_mss,speed_ms,0,blend_radius_m)
    |   movel([0.139726, -1.260671, -2.645014, -0.806705, 1.570796, 1.710523],accel_mss,speed_ms,0,blend_radius_m)
    |   movel([0.145768, -1.258827, -2.646020, -0.807543, 1.570796, 1.716564],accel_mss,speed_ms,0,blend_radius_m)
    |   movel([0.149368, -1.257783, -2.646587, -0.808018, 1.570796, 1.720164],accel_mss,speed_ms,0,blend_radius_m)
    |   movel([0.152638, -1.256876, -2.647080, -0.808433, 1.570796, 1.723434],accel_mss,speed_ms,0,blend_radius_m)
    |   movel([0.152705, -1.257095, -2.646961, -0.808333, 1.570796, 1.723501],accel_mss,speed_ms,0,blend_radius_m)
    |   movel([0.149573, -1.258165, -2.646380, -0.807844, 1.570796, 1.720369],accel_mss,speed_ms,0,blend_radius_m)
    |   movel([0.145783, -1.259381, -2.645718, -0.807290, 1.570796, 1.716579],accel_mss,speed_ms,0,blend_radius_m)
    |   movel([0.139630, -1.261300, -2.644669, -0.806420, 1.570796, 1.710426],accel_mss,speed_ms,0,blend_radius_m)
    |   movel([0.139630, -1.264321, -2.646098, -0.801970, 1.570796, 1.710426],accel_mss,speed_ms,0,blend_radius_m)
    |   movel([0.133490, -1.266214, -2.645055, -0.801121, 1.570796, 1.704286],accel_mss,speed_ms,0,blend_radius_m)
    |   movel([0.129732, -1.267339, -2.644432, -0.800618, 1.570796, 1.700529],accel_mss,speed_ms,0,blend_radius_m)
    |   movel([0.126757, -1.268210, -2.643950, -0.800229, 1.570796, 1.697554],accel_mss,speed_ms,0,blend_radius_m)
    |   movel([0.126686, -1.267995, -2.644069, -0.800325, 1.570796, 1.697483],accel_mss,speed_ms,0,blend_radius_m)
    |   movel([0.130079, -1.266791, -2.644736, -0.800862, 1.570796, 1.700875],accel_mss,speed_ms,0,blend_radius_m)
    |   movel([0.133684, -1.265599, -2.645394, -0.801396, 1.570796, 1.704480],accel_mss,speed_ms,0,blend_radius_m)
    |   movel([0.139726, -1.263692, -2.646443, -0.802254, 1.570796, 1.710523],accel_mss,speed_ms,0,blend_radius_m)
    |   movel([0.145768, -1.261851, -2.647452, -0.803086, 1.570796, 1.716564],accel_mss,speed_ms,0,blend_radius_m)
    |   movel([0.149368, -1.260809, -2.648021, -0.803558, 1.570796, 1.720164],accel_mss,speed_ms,0,blend_radius_m)
    |   movel([0.152638, -1.259904, -2.648515, -0.803970, 1.570796, 1.723434],accel_mss,speed_ms,0,blend_radius_m)
    |   movel([0.152705, -1.260122, -2.648396, -0.803871, 1.570796, 1.723501],accel_mss,speed_ms,0,blend_radius_m)
    |   movel([0.149573, -1.261191, -2.647813, -0.803385, 1.570796, 1.720369],accel_mss,speed_ms,0,blend_radius_m)
    |   movel([0.145783, -1.262405, -2.647149, -0.802835, 1.570796, 1.716579],accel_mss,speed_ms,0,blend_radius_m)
    |   movel([0.139630, -1.264321, -2.646098, -0.801970, 1.570796, 1.710426],accel_mss,speed_ms,0,blend_radius_m)
    |   movel([0.139630, -1.229499, -2.628575, -0.854315, 1.570796, 1.710426],accel_mss,speed_ms,0,blend_radius_m)
    |   speed_ms = 1.000
    |   movel([0.139340, -1.231411, -2.627571, -0.853407, 1.570796, 1.710137],accel_mss,speed_ms,0,blend_radius_m)
    |   speed_ms = 0.008
    |   movel([0.139340, -1.259601, -2.641921, -0.810867, 1.570796, 1.710137],accel_mss,speed_ms,0,blend_radius_m)
    |   speed_ms = 0.003
    |   movel([0.139340, -1.263184, -2.643635, -0.805569, 1.570796, 1.710137],accel_mss,speed_ms,0,blend_radius_m)
    |   speed_ms = 0.008
    |   movel([0.130541, -1.265922, -2.642125, -0.804342, 1.570796, 1.701337],accel_mss,speed_ms,0,blend_radius_m)
    |   movel([0.129280, -1.266301, -2.641916, -0.804173, 1.570796, 1.700076],accel_mss,speed_ms,0,blend_radius_m)
    |   movel([0.128027, -1.266651, -2.641722, -0.804016, 1.570796, 1.698823],accel_mss,speed_ms,0,blend_radius_m)
    |   movel([0.127297, -1.266823, -2.641626, -0.803940, 1.570796, 1.698093],accel_mss,speed_ms,0,blend_radius_m)
    |   movel([0.126906, -1.266893, -2.641588, -0.803908, 1.570796, 1.697702],accel_mss,speed_ms,0,blend_radius_m)
    |   movel([0.126531, -1.266904, -2.641582, -0.803904, 1.570796, 1.697328],accel_mss,speed_ms,0,blend_radius_m)
    |   movel([0.126414, -1.266629, -2.641734, -0.804026, 1.570796, 1.697211],accel_mss,speed_ms,0,blend_radius_m)
    |   movel([0.126639, -1.266273, -2.641931, -0.804185, 1.570796, 1.697435],accel_mss,speed_ms,0,blend_radius_m)
    |   movel([0.127106, -1.266016, -2.642073, -0.804300, 1.570796, 1.697902],accel_mss,speed_ms,0,blend_radius_m)
    |   movel([0.127510, -1.265838, -2.642172, -0.804379, 1.570796, 1.698306],accel_mss,speed_ms,0,blend_radius_m)
    |   movel([0.128297, -1.265530, -2.642342, -0.804517, 1.570796, 1.699094],accel_mss,speed_ms,0,blend_radius_m)
    |   movel([0.129523, -1.265099, -2.642580, -0.804710, 1.570796, 1.700319],accel_mss,speed_ms,0,blend_radius_m)
    |   movel([0.130749, -1.264692, -2.642805, -0.804892, 1.570796, 1.701545],accel_mss,speed_ms,0,blend_radius_m)
    |   movel([0.139533, -1.261929, -2.644325, -0.806136, 1.570796, 1.710330],accel_mss,speed_ms,0,blend_radius_m)
    |   movel([0.148328, -1.259241, -2.645794, -0.807354, 1.570796, 1.719124],accel_mss,speed_ms,0,blend_radius_m)
    |   movel([0.149552, -1.258889, -2.645986, -0.807514, 1.570796, 1.720349],accel_mss,speed_ms,0,blend_radius_m)
    |   movel([0.150770, -1.258563, -2.646163, -0.807662, 1.570796, 1.721566],accel_mss,speed_ms,0,blend_radius_m)
    |   movel([0.151543, -1.258388, -2.646259, -0.807743, 1.570796, 1.722340],accel_mss,speed_ms,0,blend_radius_m)
    |   movel([0.151934, -1.258320, -2.646295, -0.807773, 1.570796, 1.722730],accel_mss,speed_ms,0,blend_radius_m)
    |   movel([0.152262, -1.258279, -2.646318, -0.807792, 1.570796, 1.723058],accel_mss,speed_ms,0,blend_radius_m)
    |   movel([0.152494, -1.258440, -2.646230, -0.807719, 1.570796, 1.723290],accel_mss,speed_ms,0,blend_radius_m)
    |   movel([0.152392, -1.258810, -2.646029, -0.807550, 1.570796, 1.723188],accel_mss,speed_ms,0,blend_radius_m)
    |   movel([0.151869, -1.259165, -2.645835, -0.807388, 1.570796, 1.722666],accel_mss,speed_ms,0,blend_radius_m)
    |   movel([0.151458, -1.259344, -2.645738, -0.807307, 1.570796, 1.722255],accel_mss,speed_ms,0,blend_radius_m)
    |   movel([0.150706, -1.259631, -2.645581, -0.807176, 1.570796, 1.721502],accel_mss,speed_ms,0,blend_radius_m)
    |   movel([0.149431, -1.260064, -2.645345, -0.806980, 1.570796, 1.720227],accel_mss,speed_ms,0,blend_radius_m)
    |   movel([0.148159, -1.260469, -2.645124, -0.806796, 1.570796, 1.718955],accel_mss,speed_ms,0,blend_radius_m)
    |   movel([0.139340, -1.263184, -2.643635, -0.805569, 1.570796, 1.710137],accel_mss,speed_ms,0,blend_radius_m)
    |   movel([0.139340, -1.266202, -2.645061, -0.801126, 1.570796, 1.710137],accel_mss,speed_ms,0,blend_radius_m)
    |   movel([0.130541, -1.268935, -2.643547, -0.799907, 1.570796, 1.701337],accel_mss,speed_ms,0,blend_radius_m)
    |   movel([0.129280, -1.269313, -2.643337, -0.799739, 1.570796, 1.700076],accel_mss,speed_ms,0,blend_radius_m)
    |   movel([0.128027, -1.269662, -2.643143, -0.799584, 1.570796, 1.698823],accel_mss,speed_ms,0,blend_radius_m)
    |   movel([0.127297, -1.269835, -2.643047, -0.799507, 1.570796, 1.698093],accel_mss,speed_ms,0,blend_radius_m)
    |   movel([0.126906, -1.269904, -2.643008, -0.799476, 1.570796, 1.697702],accel_mss,speed_ms,0,blend_radius_m)
    |   movel([0.126531, -1.269915, -2.643002, -0.799472, 1.570796, 1.697328],accel_mss,speed_ms,0,blend_radius_m)
    |   movel([0.126414, -1.269641, -2.643155, -0.799593, 1.570796, 1.697211],accel_mss,speed_ms,0,blend_radius_m)
    |   movel([0.126639, -1.269286, -2.643352, -0.799751, 1.570796, 1.697435],accel_mss,speed_ms,0,blend_radius_m)
    |   movel([0.127106, -1.269029, -2.643495, -0.799865, 1.570796, 1.697902],accel_mss,speed_ms,0,blend_radius_m)
    |   movel([0.127510, -1.268851, -2.643594, -0.799944, 1.570796, 1.698306],accel_mss,speed_ms,0,blend_radius_m)
    |   movel([0.128297, -1.268544, -2.643764, -0.800081, 1.570796, 1.699094],accel_mss,speed_ms,0,blend_radius_m)
    |   movel([0.129523, -1.268114, -2.644003, -0.800272, 1.570796, 1.700319],accel_mss,speed_ms,0,blend_radius_m)
    |   movel([0.130749, -1.267707, -2.644229, -0.800454, 1.570796, 1.701545],accel_mss,speed_ms,0,blend_radius_m)
    |   movel([0.139533, -1.264948, -2.645752, -0.801688, 1.570796, 1.710330],accel_mss,speed_ms,0,blend_radius_m)
    |   movel([0.148328, -1.262265, -2.647226, -0.802898, 1.570796, 1.719124],accel_mss,speed_ms,0,blend_radius_m)
    |   movel([0.149552, -1.261914, -2.647418, -0.803057, 1.570796, 1.720349],accel_mss,speed_ms,0,blend_radius_m)
    |   movel([0.150770, -1.261589, -2.647596, -0.803205, 1.570796, 1.721566],accel_mss,speed_ms,0,blend_radius_m)
    |   movel([0.151543, -1.261413, -2.647692, -0.803284, 1.570796, 1.722340],accel_mss,speed_ms,0,blend_radius_m)
    |   movel([0.151934, -1.261346, -2.647728, -0.803315, 1.570796, 1.722730],accel_mss,speed_ms,0,blend_radius_m)
    |   movel([0.152262, -1.261305, -2.647751, -0.803334, 1.570796, 1.723058],accel_mss,speed_ms,0,blend_radius_m)
    |   movel([0.152494, -1.261466, -2.647663, -0.803261, 1.570796, 1.723290],accel_mss,speed_ms,0,blend_radius_m)
    |   movel([0.152392, -1.261835, -2.647461, -0.803093, 1.570796, 1.723188],accel_mss,speed_ms,0,blend_radius_m)
    |   movel([0.151869, -1.262189, -2.647267, -0.802933, 1.570796, 1.722666],accel_mss,speed_ms,0,blend_radius_m)
    |   movel([0.151458, -1.262368, -2.647169, -0.802852, 1.570796, 1.722255],accel_mss,speed_ms,0,blend_radius_m)
    |   movel([0.150706, -1.262655, -2.647012, -0.802722, 1.570796, 1.721502],accel_mss,speed_ms,0,blend_radius_m)
    |   movel([0.149431, -1.263087, -2.646776, -0.802527, 1.570796, 1.720227],accel_mss,speed_ms,0,blend_radius_m)
    |   movel([0.148159, -1.263491, -2.646553, -0.802344, 1.570796, 1.718955],accel_mss,speed_ms,0,blend_radius_m)
    |   movel([0.139340, -1.266202, -2.645061, -0.801126, 1.570796, 1.710137],accel_mss,speed_ms,0,blend_radius_m)
    |   movel([0.139340, -1.231411, -2.627571, -0.853407, 1.570796, 1.710137],accel_mss,speed_ms,0,blend_radius_m)
    |   speed_ms = 1.000
    |   movel([0.139005, -1.233636, -2.626398, -0.852356, 1.570796, 1.709801],accel_mss,speed_ms,0,blend_radius_m)
    |   speed_ms = 0.008
    |   movel([0.139005, -1.261797, -2.640717, -0.809875, 1.570796, 1.709801],accel_mss,speed_ms,0,blend_radius_m)
    |   speed_ms = 0.003
    |   movel([0.139005, -1.265375, -2.642427, -0.804586, 1.570796, 1.709801],accel_mss,speed_ms,0,blend_radius_m)
    |   speed_ms = 0.008
    |   movel([0.126021, -1.269439, -2.640172, -0.802778, 1.570796, 1.696818],accel_mss,speed_ms,0,blend_radius_m)
    |   movel([0.126238, -1.267891, -2.641034, -0.803464, 1.570796, 1.697034],accel_mss,speed_ms,0,blend_radius_m)
    |   movel([0.152289, -1.259836, -2.645469, -0.807083, 1.570796, 1.723085],accel_mss,speed_ms,0,blend_radius_m)
    |   movel([0.152025, -1.261417, -2.644605, -0.806367, 1.570796, 1.722822],accel_mss,speed_ms,0,blend_radius_m)
    |   movel([0.139005, -1.265375, -2.642427, -0.804586, 1.570796, 1.709801],accel_mss,speed_ms,0,blend_radius_m)
    |   movel([0.139005, -1.268389, -2.643850, -0.800149, 1.570796, 1.709801],accel_mss,speed_ms,0,blend_radius_m)
    |   movel([0.126021, -1.272446, -2.641589, -0.798354, 1.570796, 1.696818],accel_mss,speed_ms,0,blend_radius_m)
    |   movel([0.126238, -1.270901, -2.642453, -0.799036, 1.570796, 1.697034],accel_mss,speed_ms,0,blend_radius_m)
    |   movel([0.152289, -1.262860, -2.646900, -0.802629, 1.570796, 1.723085],accel_mss,speed_ms,0,blend_radius_m)
    |   movel([0.152025, -1.264438, -2.646033, -0.801918, 1.570796, 1.722822],accel_mss,speed_ms,0,blend_radius_m)
    |   movel([0.139005, -1.268389, -2.643850, -0.800149, 1.570796, 1.709801],accel_mss,speed_ms,0,blend_radius_m)
    |   movel([0.139005, -1.233636, -2.626398, -0.852356, 1.570796, 1.709801],accel_mss,speed_ms,0,blend_radius_m)
    |   speed_ms = 1.000
    |   movel([0.138813, -1.234903, -2.625726, -0.851759, 1.570796, 1.709610],accel_mss,speed_ms,0,blend_radius_m)
    |   speed_ms = 0.008
    |   movel([0.138813, -1.263048, -2.640028, -0.809313, 1.570796, 1.709610],accel_mss,speed_ms,0,blend_radius_m)
    |   speed_ms = 0.003
    |   movel([0.138813, -1.266624, -2.641737, -0.804028, 1.570796, 1.709610],accel_mss,speed_ms,0,blend_radius_m)
    |   speed_ms = 0.008
    |   movel([0.132711, -1.268494, -2.640698, -0.803196, 1.570796, 1.703507],accel_mss,speed_ms,0,blend_radius_m)
    |   movel([0.128976, -1.269606, -2.640079, -0.802704, 1.570796, 1.699772],accel_mss,speed_ms,0,blend_radius_m)
    |   movel([0.126019, -1.270466, -2.639599, -0.802324, 1.570796, 1.696815],accel_mss,speed_ms,0,blend_radius_m)
    |   movel([0.125948, -1.270252, -2.639718, -0.802419, 1.570796, 1.696745],accel_mss,speed_ms,0,blend_radius_m)
    |   movel([0.129320, -1.269061, -2.640383, -0.802945, 1.570796, 1.700116],accel_mss,speed_ms,0,blend_radius_m)
    |   movel([0.132903, -1.267883, -2.641038, -0.803468, 1.570796, 1.703700],accel_mss,speed_ms,0,blend_radius_m)
    |   movel([0.138909, -1.266000, -2.642082, -0.804307, 1.570796, 1.709705],accel_mss,speed_ms,0,blend_radius_m)
    |   movel([0.144913, -1.264182, -2.643086, -0.805121, 1.570796, 1.715709],accel_mss,speed_ms,0,blend_radius_m)
    |   movel([0.148491, -1.263153, -2.643652, -0.805583, 1.570796, 1.719288],accel_mss,speed_ms,0,blend_radius_m)
    |   movel([0.151741, -1.262259, -2.644143, -0.805986, 1.570796, 1.722538],accel_mss,speed_ms,0,blend_radius_m)
    |   movel([0.151808, -1.262476, -2.644024, -0.805888, 1.570796, 1.722605],accel_mss,speed_ms,0,blend_radius_m)
    |   movel([0.148695, -1.263533, -2.643444, -0.805413, 1.570796, 1.719492],accel_mss,speed_ms,0,blend_radius_m)
    |   movel([0.144929, -1.264732, -2.642783, -0.804874, 1.570796, 1.715725],accel_mss,speed_ms,0,blend_radius_m)
    |   movel([0.138813, -1.266624, -2.641737, -0.804028, 1.570796, 1.709610],accel_mss,speed_ms,0,blend_radius_m)
    |   movel([0.138813, -1.269636, -2.643157, -0.799595, 1.570796, 1.709610],accel_mss,speed_ms,0,blend_radius_m)
    |   movel([0.132711, -1.271503, -2.642117, -0.798770, 1.570796, 1.703507],accel_mss,speed_ms,0,blend_radius_m)
    |   movel([0.128976, -1.272612, -2.641496, -0.798281, 1.570796, 1.699772],accel_mss,speed_ms,0,blend_radius_m)
    |   movel([0.126019, -1.273471, -2.641014, -0.797904, 1.570796, 1.696815],accel_mss,speed_ms,0,blend_radius_m)
    |   movel([0.125948, -1.273258, -2.641134, -0.797997, 1.570796, 1.696745],accel_mss,speed_ms,0,blend_radius_m)
    |   movel([0.129320, -1.272069, -2.641800, -0.798520, 1.570796, 1.700116],accel_mss,speed_ms,0,blend_radius_m)
    |   movel([0.132903, -1.270893, -2.642457, -0.799039, 1.570796, 1.703700],accel_mss,speed_ms,0,blend_radius_m)
    |   movel([0.138909, -1.269013, -2.643504, -0.799872, 1.570796, 1.709705],accel_mss,speed_ms,0,blend_radius_m)
    |   movel([0.144913, -1.267198, -2.644511, -0.800681, 1.570796, 1.715709],accel_mss,speed_ms,0,blend_radius_m)
    |   movel([0.148491, -1.266171, -2.645078, -0.801140, 1.570796, 1.719288],accel_mss,speed_ms,0,blend_radius_m)
    |   movel([0.151741, -1.265278, -2.645571, -0.801540, 1.570796, 1.722538],accel_mss,speed_ms,0,blend_radius_m)
    |   movel([0.151808, -1.265495, -2.645451, -0.801443, 1.570796, 1.722605],accel_mss,speed_ms,0,blend_radius_m)
    |   movel([0.148695, -1.266550, -2.644869, -0.800970, 1.570796, 1.719492],accel_mss,speed_ms,0,blend_radius_m)
    |   movel([0.144929, -1.267747, -2.644207, -0.800436, 1.570796, 1.715725],accel_mss,speed_ms,0,blend_radius_m)
    |   movel([0.138813, -1.269636, -2.643157, -0.799595, 1.570796, 1.709610],accel_mss,speed_ms,0,blend_radius_m)
    |   movel([0.138813, -1.234903, -2.625726, -0.851759, 1.570796, 1.709610],accel_mss,speed_ms,0,blend_radius_m)
    |   speed_ms = 1.000
    |   movel([0.138813, -1.141047, -2.563360, -1.007982, 1.570796, 1.709610],accel_mss,speed_ms,0,blend_radius_m)
    |   # End of main program
    | end
    | 
    | Machining3()
